	{attribute 'c++_compatible'}
	{attribute 'external_name' := 'FB_VN_ReadRegister_ULINT_GUID_0511260A_434E_4D8A_DC8D_C67C5FC0DC86'}
	{attribute 'TcIecLibraryType'}
	(* This FB reads a ULINT register from the camera. Requires an open control channel (e.g. by calling FB_VN_GevCameraControl.OpenCamera() before) *)
	FUNCTION_BLOCK FB_VN_ReadRegister_ULINT
	VAR_INPUT
		(* The address of the register that should be read *)
		 {attribute 'GUID' := 'E1ED2436-3512-43FA-B927-3F71DEDDA853'}
		nAddress : GVCP_REGISTER_ADDRESS;
		(* OPTIONAL: The endianness of the register. 0 = Big, 1 = Little. Default: 0 *)
		nEndian : UINT;
		(* Reading the register is triggered by a rising edge at this input. *)
		bRead : BOOL;
	END_VAR
	VAR
		 {attribute 'hide'}
		_reserved1 : USINT;
	END_VAR
	VAR_INPUT
		(* Indicates the time before the function is cancelled. *)
		nTimeout : TIME := VISION_ADS_TIMEOUT;
	END_VAR
	VAR
		 {attribute 'hide'}
		_reserved2 : UINT_0_32;
	END_VAR
	VAR_OUTPUT
		(* The read value *)
		nValue : ULINT;
		(* This output remains TRUE until the function block has executed a command, but at the longest for the duration supplied to the 'nTimeout' input. While bBusy = TRUE, no new command will be accepted at the inputs. *)
		bBusy : BOOL;
		(* This output is switched to TRUE as soon as an error occurs during the execution of a command. The command-specific error code is contained in ‘nErrorId’. If the function block has a timeout error, 'bError' is TRUE and 'nErrorId' is 1861 (hexadecimal 0x745). Is reset to FALSE by the execution of a command at the inputs. *)
		bError : BOOL;
	END_VAR
	VAR
		 {attribute 'hide'}
		_reserved3 : UINT;
	END_VAR
	VAR_OUTPUT
		(* Contains the ADS error code or the command-specific error code of the last executed command. Is reset to 0 by the execution of a command at the inputs. *)
		nErrorId : UDINT;
	END_VAR
	VAR
		(* Internal reference to the corresponding TcVnGevImageProvider TcCOM module ID, which needs to be set via TC init symbol. *)
		{attribute 'TcInitSymbol'}
		{attribute 'TcCategoryOID' := 'TcVnGevImageProvider'}
		 {attribute 'GUID' := '18071995-0000-0000-0000-00000000000F'}
		oidITcVnGevImageProvider : OTCID;
		 {attribute 'hide'}
		_reserved4 : UINT_0_32;
		(* Internal reference to the corresponding TcVnGevImageProvider module. *)
		{attribute 'hide'}
		 {attribute 'GUID' := 'ED7659DB-95DC-4A4A-B62F-02C9870D5E81'}
		ipGevImageProvider : ITcVnGevImageProvider;
		(* Internal timestamp for timeout detection *)
		{attribute 'hide'}
		nTimeElapsed : TIME;
		(* Internal flag for rising edge detection *)
		{attribute 'hide'}
		bLastRead : BOOL;
		 {attribute 'hide'}
		_reserved5 : ARRAY [1..3] OF USINT;
	END_VAR


	(* Internal method *)
	{attribute 'hide'}
	METHOD FB_exit : BOOL
	VAR_INPUT
		(*  if TRUE, the exit method is called for exiting an instance that is copied afterwards (online change). *)
		bInCopyCode : BOOL;
	END_VAR
END_METHOD


	(* Internal method *)
	{attribute 'hide'}
	METHOD FB_init : BOOL
	VAR_INPUT
		(*  if TRUE, the retain variables are initialized (warm start / cold start) *)
		bInitRetains : BOOL;
		(*  if TRUE, the instance afterwards gets moved into the copy code (online change) *)
		bInCopyCode : BOOL;
	END_VAR
END_METHOD

END_FUNCTION_BLOCK

// Function Blocks/Camera Register Access/FB_VN_WriteRegister_ULINT

	{attribute 'c++_compatible'}
	{attribute 'external_name' := 'FB_VN_WriteRegister_ULINT_GUID_9D472D1C_82B4_4199_F5A1_B64D0453F3B0'}
	{attribute 'TcIecLibraryType'}
	(* This FB writes a ULINT value into a register on the camera. Requires an open control channel (e.g. by calling FB_VN_GevCameraControl.OpenCamera() before) *)
	FUNCTION_BLOCK FB_VN_WriteRegister_ULINT
	VAR_INPUT
		(* The address of the register that should be written *)
		 {attribute 'GUID' := 'E1ED2436-3512-43FA-B927-3F71DEDDA853'}
		nAddress : GVCP_REGISTER_ADDRESS;
	END_VAR
	VAR
		 {attribute 'hide'}
		_reserved1 : UINT_0_32;
	END_VAR
	VAR_INPUT
		(* The value to write *)
		nValue : ULINT;
		(* OPTIONAL: The endianness of the register. 0 = Big, 1 = Little. Default: 0 *)
		nEndian : UINT;
		(* Writing the register is triggered by a rising edge at this input. *)
		bWrite : BOOL;
	END_VAR
	VAR
		 {attribute 'hide'}
		_reserved2 : USINT;
	END_VAR
	VAR_INPUT
		(* Indicates the time before the function is cancelled. *)
		nTimeout : TIME := VISION_ADS_TIMEOUT;
	END_VAR
	VAR_OUTPUT
		(* This output remains TRUE until the function block has executed a command, but at the longest for the duration supplied to the 'nTimeout' input. While bBusy = TRUE, no new command will be accepted at the inputs. *)
		bBusy : BOOL;
		(* This output is switched to TRUE as soon as an error occurs during the execution of a command. The command-specific error code is contained in ‘nErrorId’. If the function block has a timeout error, 'bError' is TRUE and 'nErrorId' is 1861 (hexadecimal 0x745). Is reset to FALSE by the execution of a command at the inputs. *)
		bError : BOOL;
	END_VAR
	VAR
		 {attribute 'hide'}
		_reserved3 : UINT;
	END_VAR
	VAR_OUTPUT
		(* Contains the ADS error code or the command-specific error code of the last executed command. Is reset to 0 by the execution of a command at the inputs. *)
		nErrorId : UDINT;
	END_VAR
	VAR
		(* Internal reference to the corresponding TcVnGevImageProvider TcCOM module ID, which needs to be set via TC init symbol. *)
		{attribute 'TcInitSymbol'}
		{attribute 'TcCategoryOID' := 'TcVnGevImageProvider'}
		 {attribute 'GUID' := '18071995-0000-0000-0000-00000000000F'}
		oidITcVnGevImageProvider : OTCID;
		 {attribute 'hide'}
		_reserved4 : UINT_0_32;
		(* Internal reference to the corresponding TcVnGevImageProvider module. *)
		{attribute 'hide'}
		 {attribute 'GUID' := 'ED7659DB-95DC-4A4A-B62F-02C9870D5E81'}
		ipGevImageProvider : ITcVnGevImageProvider;
		(* Internal timestamp for timeout detection *)
		{attribute 'hide'}
		nTimeElapsed : TIME;
		(* Internal flag for rising edge detection *)
		{attribute 'hide'}
		bLastWrite : BOOL;
		 {attribute 'hide'}
		_reserved5 : ARRAY [1..3] OF USINT;
	END_VAR


	(* Internal method *)
	{attribute 'hide'}
	METHOD FB_exit : BOOL
	VAR_INPUT
		(*  if TRUE, the exit method is called for exiting an instance that is copied afterwards (online change). *)
		bInCopyCode : BOOL;
	END_VAR
END_METHOD


	(* Internal method *)
	{attribute 'hide'}
	METHOD FB_init : BOOL
	VAR_INPUT
		(*  if TRUE, the retain variables are initialized (warm start / cold start) *)
		bInitRetains : BOOL;
		(*  if TRUE, the instance afterwards gets moved into the copy code (online change) *)
		bInCopyCode : BOOL;
	END_VAR
END_METHOD

END_FUNCTION_BLOCK

// Function Blocks/Camera Register Access/FB_VN_ReadMemory

	{attribute 'c++_compatible'}
	{attribute 'external_name' := 'FB_VN_ReadMemory_GUID_F43A0502_950A_4FC1_EE1B_7AC9DA03F230'}
	{attribute 'TcIecLibraryType'}
	(* This FB reads consecutive memory locations from the camera. Requires an open control channel (e.g. by calling FB_VN_GevCameraControl.OpenCamera() before) *)
	FUNCTION_BLOCK FB_VN_ReadMemory
	VAR_INPUT
		(* The address of the first byte to read from the camera (must be 32-bit aligned) *)
		 {attribute 'GUID' := 'E1ED2436-3512-43FA-B927-3F71DEDDA853'}
		nAddress : GVCP_REGISTER_ADDRESS;
		(* The number of bytes to read, starting with nAddress (must be a multiple of 4, not more than 536) *)
		nLength : UINT;
	END_VAR
	VAR
		 {attribute 'hide'}
		_reserved1 : UINT;
	END_VAR
	VAR_INPUT
		(* Pointer to the buffer where the read memory content is written to (The buffer must have a size of at least nLength bytes!) *)
		 {attribute 'GUID' := '18071995-0000-0000-0000-000000000018'}
		pBuffer : PVOID;
		(* Reading the memory is triggered by a rising edge at this input. *)
		bRead : BOOL;
	END_VAR
	VAR
		 {attribute 'hide'}
		_reserved2 : ARRAY [1..3] OF USINT;
	END_VAR
	VAR_INPUT
		(* Indicates the time before the function is cancelled. *)
		nTimeout : TIME := VISION_ADS_TIMEOUT;
	END_VAR
	VAR_OUTPUT
		(* This output remains TRUE until the function block has executed a command, but at the longest for the duration supplied to the 'nTimeout' input. While bBusy = TRUE, no new command will be accepted at the inputs. *)
		bBusy : BOOL;
		(* This output is switched to TRUE as soon as an error occurs during the execution of a command. The command-specific error code is contained in ‘nErrorId’. If the function block has a timeout error, 'bError' is TRUE and 'nErrorId' is 1861 (hexadecimal 0x745). Is reset to FALSE by the execution of a command at the inputs. *)
		bError : BOOL;
	END_VAR
	VAR
		 {attribute 'hide'}
		_reserved3 : UINT;
	END_VAR
	VAR_OUTPUT
		(* Contains the ADS error code or the command-specific error code of the last executed command. Is reset to 0 by the execution of a command at the inputs. *)
		nErrorId : UDINT;
	END_VAR
	VAR
		(* Internal reference to the corresponding TcVnGevImageProvider TcCOM module ID, which needs to be set via TC init symbol. *)
		{attribute 'TcInitSymbol'}
		{attribute 'TcCategoryOID' := 'TcVnGevImageProvider'}
		 {attribute 'GUID' := '18071995-0000-0000-0000-00000000000F'}
		oidITcVnGevImageProvider : OTCID;
		 {attribute 'hide'}
		_reserved4 : UINT_0_32;
		(* Internal reference to the corresponding TcVnGevImageProvider module. *)
		{attribute 'hide'}
		 {attribute 'GUID' := 'ED7659DB-95DC-4A4A-B62F-02C9870D5E81'}
		ipGevImageProvider : ITcVnGevImageProvider;
		(* Internal timestamp for timeout detection *)
		{attribute 'hide'}
		nTimeElapsed : TIME;
		(* Internal flag for rising edge detection *)
		{attribute 'hide'}
		bLastRead : BOOL;
		 {attribute 'hide'}
		_reserved5 : ARRAY [1..3] OF USINT;
	END_VAR


	(* Internal method *)
	{attribute 'hide'}
	METHOD FB_exit : BOOL
	VAR_INPUT
		(* If TRUE, the exit method is called for exiting an instance that is copied afterwards (online change). *)
		bInCopyCode : BOOL;
	END_VAR
END_METHOD


	(* Internal method *)
	{attribute 'hide'}
	METHOD FB_init : BOOL
	VAR_INPUT
		(* If TRUE, the retain variables are initialized (warm start / cold start) *)
		bInitRetains : BOOL;
		(* If TRUE, the instance afterwards gets moved into the copy code (online change) *)
		bInCopyCode : BOOL;
	END_VAR
END_METHOD

END_FUNCTION_BLOCK

// Function Blocks/Camera Register Access/FB_VN_WriteMemory

	{attribute 'c++_compatible'}
	{attribute 'external_name' := 'FB_VN_WriteMemory_GUID_E11A1718_DC13_44E5_FD90_B3F294477065'}
	{attribute 'TcIecLibraryType'}
	(* This FB writes data to consecutive memory locations on the camera. Requires an open control channel (e.g. by calling FB_VN_GevCameraControl.OpenCamera() before) *)
	FUNCTION_BLOCK FB_VN_WriteMemory
	VAR_INPUT
		(* The address of the first byte to write to the camera (must be 32-bit aligned) *)
		 {attribute 'GUID' := 'E1ED2436-3512-43FA-B927-3F71DEDDA853'}
		nAddress : GVCP_REGISTER_ADDRESS;
		(* The number of bytes to write, starting at nAddress (must be a multiple of 4, not more than 536) *)
		nLength : UINT;
	END_VAR
	VAR
		 {attribute 'hide'}
		_reserved1 : UINT;
	END_VAR
	VAR_INPUT
		(* Pointer to the data that should be written to the camera (must have a size of at least nLength bytes!) *)
		 {attribute 'GUID' := '18071995-0000-0000-0000-000000000018'}
		pData : PVOID;
		(* Writing the memory is triggered by a rising edge at this input. *)
		bWrite : BOOL;
	END_VAR
	VAR
		 {attribute 'hide'}
		_reserved2 : ARRAY [1..3] OF USINT;
	END_VAR
	VAR_INPUT
		(* Indicates the time before the function is cancelled. *)
		nTimeout : TIME := VISION_ADS_TIMEOUT;
	END_VAR
	VAR_OUTPUT
		(* This output remains TRUE until the function block has executed a command, but at the longest for the duration supplied to the 'nTimeout' input. While bBusy = TRUE, no new command will be accepted at the inputs. *)
		bBusy : BOOL;
		(* This output is switched to TRUE as soon as an error occurs during the execution of a command. The command-specific error code is contained in ‘nErrorId’. If the function block has a timeout error, 'bError' is TRUE and 'nErrorId' is 1861 (hexadecimal 0x745). Is reset to FALSE by the execution of a command at the inputs. *)
		bError : BOOL;
	END_VAR
	VAR
		 {attribute 'hide'}
		_reserved3 : UINT;
	END_VAR
	VAR_OUTPUT
		(* Contains the ADS error code or the command-specific error code of the last executed command. Is reset to 0 by the execution of a command at the inputs. *)
		nErrorId : UDINT;
		(* The number of bytes that have been successfully written to the camera. *)
		nBytesWritten : UINT;
	END_VAR
	VAR
		 {attribute 'hide'}
		_reserved4 : UINT;
		(* Internal reference to the corresponding TcVnGevImageProvider TcCOM module ID, which needs to be set via TC init symbol. *)
		{attribute 'TcInitSymbol'}
		{attribute 'TcCategoryOID' := 'TcVnGevImageProvider'}
		 {attribute 'GUID' := '18071995-0000-0000-0000-00000000000F'}
		oidITcVnGevImageProvider : OTCID;
		(* Internal reference to the corresponding TcVnGevImageProvider module. *)
		{attribute 'hide'}
		 {attribute 'GUID' := 'ED7659DB-95DC-4A4A-B62F-02C9870D5E81'}
		ipGevImageProvider : ITcVnGevImageProvider;
		(* Internal timestamp for timeout detection *)
		{attribute 'hide'}
		nTimeElapsed : TIME;
		(* Internal flag for rising edge detection *)
		{attribute 'hide'}
		bLastRead : BOOL;
		 {attribute 'hide'}
		_reserved5 : ARRAY [1..3] OF USINT;
	END_VAR


	(* Internal method *)
	{attribute 'hide'}
	METHOD FB_exit : BOOL
	VAR_INPUT
		(* If TRUE, the exit method is called for exiting an instance that is copied afterwards (online change). *)
		bInCopyCode : BOOL;
	END_VAR
END_METHOD


	(* Internal method *)
	{attribute 'hide'}
	METHOD FB_init : BOOL
	VAR_INPUT
		(* If TRUE, the retain variables are initialized (warm start / cold start) *)
		bInitRetains : BOOL;
		(* If TRUE, the instance afterwards gets moved into the copy code (online change) *)
		bInCopyCode : BOOL;
	END_VAR
END_METHOD

END_FUNCTION_BLOCK

// Function Blocks/Camera Register Access/FB_VN_ReadRegister_REAL

	{attribute 'c++_compatible'}
	{attribute 'external_name' := 'FB_VN_ReadRegister_REAL_GUID_8300240C_129D_40AD_E145_72F0B3958AC0'}
	{attribute 'TcIecLibraryType'}
	(* This FB reads a REAL register from the camera. Requires an open control channel (e.g. by calling FB_VN_GevCameraControl.OpenCamera() before) *)
	FUNCTION_BLOCK FB_VN_ReadRegister_REAL
	VAR_INPUT
		(* The address of the register that should be read *)
		 {attribute 'GUID' := 'E1ED2436-3512-43FA-B927-3F71DEDDA853'}
		nAddress : GVCP_REGISTER_ADDRESS;
		(* OPTIONAL: The endianness of the register. 0 = Big, 1 = Little. Default: 0 *)
		nEndian : UINT;
		(* Reading the register is triggered by a rising edge at this input. *)
		bRead : BOOL;
	END_VAR
	VAR
		 {attribute 'hide'}
		_reserved1 : USINT;
	END_VAR
	VAR_INPUT
		(* Indicates the time before the function is cancelled. *)
		nTimeout : TIME := VISION_ADS_TIMEOUT;
	END_VAR
	VAR_OUTPUT
		(* The read value *)
		fValue : REAL;
		(* This output remains TRUE until the function block has executed a command, but at the longest for the duration supplied to the 'nTimeout' input. While bBusy = TRUE, no new command will be accepted at the inputs. *)
		bBusy : BOOL;
		(* This output is switched to TRUE as soon as an error occurs during the execution of a command. The command-specific error code is contained in ‘nErrorId’. If the function block has a timeout error, 'bError' is TRUE and 'nErrorId' is 1861 (hexadecimal 0x745). Is reset to FALSE by the execution of a command at the inputs. *)
		bError : BOOL;
	END_VAR
	VAR
		 {attribute 'hide'}
		_reserved2 : UINT;
	END_VAR
	VAR_OUTPUT
		(* Contains the ADS error code or the command-specific error code of the last executed command. Is reset to 0 by the execution of a command at the inputs. *)
		nErrorId : UDINT;
	END_VAR
	VAR
		(* Internal reference to the corresponding TcVnGevImageProvider TcCOM module ID, which needs to be set via TC init symbol. *)
		{attribute 'TcInitSymbol'}
		{attribute 'TcCategoryOID' := 'TcVnGevImageProvider'}
		 {attribute 'GUID' := '18071995-0000-0000-0000-00000000000F'}
		oidITcVnGevImageProvider : OTCID;
		 {attribute 'hide'}
		_reserved3 : UINT_0_32;
		(* Internal reference to the corresponding TcVnGevImageProvider module. *)
		{attribute 'hide'}
		 {attribute 'GUID' := 'ED7659DB-95DC-4A4A-B62F-02C9870D5E81'}
		ipGevImageProvider : ITcVnGevImageProvider;
		(* Internal timestamp for timeout detection *)
		{attribute 'hide'}
		nTimeElapsed : TIME;
		(* Internal flag for rising edge detection *)
		{attribute 'hide'}
		bLastRead : BOOL;
		 {attribute 'hide'}
		_reserved4 : ARRAY [1..3] OF USINT;
	END_VAR


	(* Internal method *)
	{attribute 'hide'}
	METHOD FB_exit : BOOL
	VAR_INPUT
		(*  if TRUE, the exit method is called for exiting an instance that is copied afterwards (online change). *)
		bInCopyCode : BOOL;
	END_VAR
END_METHOD


	(* Internal method *)
	{attribute 'hide'}
	METHOD FB_init : BOOL
	VAR_INPUT
		(*  if TRUE, the retain variables are initialized (warm start / cold start) *)
		bInitRetains : BOOL;
		(*  if TRUE, the instance afterwards gets moved into the copy code (online change) *)
		bInCopyCode : BOOL;
	END_VAR
END_METHOD

END_FUNCTION_BLOCK

// Function Blocks/Camera Register Access/FB_VN_WriteRegister_REAL

	{attribute 'c++_compatible'}
	{attribute 'external_name' := 'FB_VN_WriteRegister_REAL_GUID_9406F075_95E1_49DE_E4AE_6ECDFB627AD5'}
	{attribute 'TcIecLibraryType'}
	(* This FB writes a REAL value into a register on the camera. Requires an open control channel (e.g. by calling FB_VN_GevCameraControl.OpenCamera() before) *)
	FUNCTION_BLOCK FB_VN_WriteRegister_REAL
	VAR_INPUT
		(* The address of the register that should be written *)
		 {attribute 'GUID' := 'E1ED2436-3512-43FA-B927-3F71DEDDA853'}
		nAddress : GVCP_REGISTER_ADDRESS;
		(* The value to write *)
		fValue : REAL;
		(* OPTIONAL: The endianness of the register. 0 = Big, 1 = Little. Default: 0 *)
		nEndian : UINT;
		(* Writing the register is triggered by a rising edge at this input. *)
		bWrite : BOOL;
	END_VAR
	VAR
		 {attribute 'hide'}
		_reserved1 : USINT;
	END_VAR
	VAR_INPUT
		(* Indicates the time before the function is cancelled. *)
		nTimeout : TIME := VISION_ADS_TIMEOUT;
	END_VAR
	VAR_OUTPUT
		(* This output remains TRUE until the function block has executed a command, but at the longest for the duration supplied to the 'nTimeout' input. While bBusy = TRUE, no new command will be accepted at the inputs. *)
		bBusy : BOOL;
		(* This output is switched to TRUE as soon as an error occurs during the execution of a command. The command-specific error code is contained in ‘nErrorId’. If the function block has a timeout error, 'bError' is TRUE and 'nErrorId' is 1861 (hexadecimal 0x745). Is reset to FALSE by the execution of a command at the inputs. *)
		bError : BOOL;
	END_VAR
	VAR
		 {attribute 'hide'}
		_reserved2 : UINT;
	END_VAR
	VAR_OUTPUT
		(* Contains the ADS error code or the command-specific error code of the last executed command. Is reset to 0 by the execution of a command at the inputs. *)
		nErrorId : UDINT;
	END_VAR
	VAR
		(* Internal reference to the corresponding TcVnGevImageProvider TcCOM module ID, which needs to be set via TC init symbol. *)
		{attribute 'TcInitSymbol'}
		{attribute 'TcCategoryOID' := 'TcVnGevImageProvider'}
		 {attribute 'GUID' := '18071995-0000-0000-0000-00000000000F'}
		oidITcVnGevImageProvider : OTCID;
		 {attribute 'hide'}
		_reserved3 : UINT_0_32;
		(* Internal reference to the corresponding TcVnGevImageProvider module. *)
		{attribute 'hide'}
		 {attribute 'GUID' := 'ED7659DB-95DC-4A4A-B62F-02C9870D5E81'}
		ipGevImageProvider : ITcVnGevImageProvider;
		(* Internal timestamp for timeout detection *)
		{attribute 'hide'}
		nTimeElapsed : TIME;
		(* Internal flag for rising edge detection *)
		{attribute 'hide'}
		bLastWrite : BOOL;
		 {attribute 'hide'}
		_reserved4 : ARRAY [1..3] OF USINT;
	END_VAR


	(* Internal method *)
	{attribute 'hide'}
	METHOD FB_exit : BOOL
	VAR_INPUT
		(*  if TRUE, the exit method is called for exiting an instance that is copied afterwards (online change). *)
		bInCopyCode : BOOL;
	END_VAR
END_METHOD


	(* Internal method *)
	{attribute 'hide'}
	METHOD FB_init : BOOL
	VAR_INPUT
		(*  if TRUE, the retain variables are initialized (warm start / cold start) *)
		bInitRetains : BOOL;
		(*  if TRUE, the instance afterwards gets moved into the copy code (online change) *)
		bInCopyCode : BOOL;
	END_VAR
END_METHOD

END_FUNCTION_BLOCK

// Function Blocks/Image Processing/FB_VN_GeneralizedHoughBallard

	{attribute 'c++_compatible'}
	{attribute 'external_name' := 'FB_VN_GeneralizedHoughBallard_GUID_A0476776_FAE7_4198_C858_300BFA209DB8'}
	{attribute 'TcIecLibraryType'}
	{attribute 'no_explicit_call' :='do not call this POU directly'}
	(* This FB provides the Generalized Hough Ballard functionality. First, set the parameters via the corresponding methods (optional, defaults are used otherwise). Then, set the template (required). Afterwards, the Detect method can be executed. *)
	FUNCTION_BLOCK FB_VN_GeneralizedHoughBallard
	VAR
		(* Internal stuff *)
		{attribute 'hide'}
		 {attribute 'GUID' := '18071995-0000-0000-0000-000000000018'}
		internal1 : PVOID;
		(* Internal stuff *)
		{attribute 'hide'}
		 {attribute 'GUID' := '18071995-0000-0000-0000-000000000018'}
		internal2 : PVOID;
		(* Internal stuff *)
		{attribute 'hide'}
		internal3 : BOOL;
		 {attribute 'hide'}
		_reserved1 : UINT_24_56;
	END_VAR


	(* Internal method *)
	{attribute 'hide'}
	METHOD FB_exit : BOOL
	VAR_INPUT
		(* if TRUE, the exit method is called for exiting an instance that is copied afterwards (online change). *)
		bInCopyCode : BOOL;
	END_VAR
END_METHOD


	(* Internal method *)
	{attribute 'hide'}
	METHOD FB_init : BOOL
	VAR_INPUT
		(* if TRUE, the retain variables are initialized (warm start / cold start) *)
		bInitRetains : BOOL;
		(* if TRUE, the instance afterwards gets moved into the copy code (online change) *)
		bInCopyCode : BOOL;
	END_VAR
END_METHOD


	(* Detect the template in an image (SetTemplate must have been called before). *)
	METHOD Detect : HRESULT
	VAR_INPUT
		(* Source image (1 channel, USINT) *)
 {attribute 'GUID' := '70D42C6D-6F4E-4719-8B29-2883D5D59B1C'}
				ipImage : ITcVnImage;
		(* Returns the centers of the detected template positions (ContainerType_Vector_TcVnPoint2_REAL; Non-zero interface pointers are reused.) *)
 {attribute 'GUID' := 'BC72B333-E095-465B-9693-7979773CA3B8'}
				ipPositions : REFERENCE TO ITcVnContainer;
	END_VAR
END_METHOD


	(* Sets the canny edge detection thresholds. *)
	METHOD SetCannyThreshold : HRESULT
	VAR_INPUT
		(* Low threshold (> 0) *)
		nLow : DINT;
		(* High threshold (> nLow, usually 2 to 3 * nLow) *)
		nHigh : DINT;
	END_VAR
END_METHOD


	(* Sets the inverted ratio of the accumulator size in relation to the source image's size (e.g. a value of 2 means that the size is halved in both directions.) *)
	METHOD SetInvAccuRatio : HRESULT
	VAR_INPUT
		(* Inverted accumulator ratio (> 0) *)
		fInvAccuRatio : LREAL;
	END_VAR
END_METHOD


	(* Sets the number of R-table levels. *)
	METHOD SetLevels : HRESULT
	VAR_INPUT
		(* Number of R-table levels (> 0) *)
		nLevels : DINT;
	END_VAR
END_METHOD


	(* Sets the minimum distance between the centers of different objects. *)
	METHOD SetMinDist : HRESULT
	VAR_INPUT
		(* Minimum distance (> 0) *)
		fMinDist : LREAL;
	END_VAR
END_METHOD


	(* Sets the template image to search for in the Detect method. *)
	METHOD SetTemplate : HRESULT
	VAR_INPUT
		(* Template image (1 channel, USINT) *)
 {attribute 'GUID' := '70D42C6D-6F4E-4719-8B29-2883D5D59B1C'}
				ipImage : ITcVnImage;
	END_VAR
END_METHOD


	(* Sets the accumulator threshold, i.e. the number of votes required to detect a match (too small values lead to false detections). *)
	METHOD SetVotesThreshold : HRESULT
	VAR_INPUT
		(* Number of votes required to detect a match (> 0) *)
		nVotes : DINT;
	END_VAR
END_METHOD

END_FUNCTION_BLOCK

// Function Blocks/Image Processing/FB_VN_SSIM

	{attribute 'c++_compatible'}
	{attribute 'external_name' := 'FB_VN_SSIM_GUID_4075B8D8_49BB_4B5C_CD74_E48AAA73AD77'}
	{attribute 'TcIecLibraryType'}
	{attribute 'no_explicit_call' :='do not call this POU directly'}
	(* This FB provides the structural similarity (SSIM) functionality. First, set the reference image. Afterwards, the Compute method can be executed. *)
	FUNCTION_BLOCK FB_VN_SSIM
	VAR
		(* Internal stuff *)
		{attribute 'hide'}
		 {attribute 'GUID' := '18071995-0000-0000-0000-000000000018'}
		internal1 : PVOID;
	END_VAR


	(* Internal method *)
	{attribute 'hide'}
	METHOD FB_exit : BOOL
	VAR_INPUT
		(* if TRUE, the exit method is called for exiting an instance that is copied afterwards (online change). *)
		bInCopyCode : BOOL;
	END_VAR
END_METHOD


	(* Internal method *)
	{attribute 'hide'}
	METHOD FB_init : BOOL
	VAR_INPUT
		(* if TRUE, the retain variables are initialized (warm start / cold start) *)
		bInitRetains : BOOL;
		(* if TRUE, the instance afterwards gets moved into the copy code (online change) *)
		bInCopyCode : BOOL;
	END_VAR
END_METHOD


	(* Compute the structural similarity (SetReference must have been called before). *)
	METHOD Compute : HRESULT
	VAR_INPUT
		(* Source image (USINT) *)
 {attribute 'GUID' := '70D42C6D-6F4E-4719-8B29-2883D5D59B1C'}
				ipSrcImage : ITcVnImage;
		(* Returns the SSIM (REAL, values from 0 to 1) *)
 {attribute 'GUID' := '70D42C6D-6F4E-4719-8B29-2883D5D59B1C'}
				ipSSIM : REFERENCE TO ITcVnImage;
	END_VAR
END_METHOD


	(* Sets the reference image, used by the SSIM method. *)
	METHOD SetReference : HRESULT
	VAR_INPUT
		(* Reference image (USINT) *)
 {attribute 'GUID' := '70D42C6D-6F4E-4719-8B29-2883D5D59B1C'}
				ipImage : ITcVnImage;
	END_VAR
END_METHOD

END_FUNCTION_BLOCK

// Functions/Control Functions/F_VN_StartAbsWatchdog

	{attribute 'TcIecLibraryType'}
	{attribute 'external_name' := 'F_VN_StartAbsWatchdog_GUID_354F303E_246D_4234_D496_3202655F920B'}
	(* Starts a cooperative watchdog given an absolute stop time. *)
	FUNCTION F_VN_StartAbsWatchdog : HRESULT
	VAR_INPUT
		tStop	:	DINT;	(* Stop time in us *)
		hrPrev	:	HRESULT;	(* HRESULT indicating the result of previous operations (If SUCCEEDED(hrPrev) equals false, no operation is executed.) *)
	END_VAR

END_FUNCTION

// Functions/Control Functions/F_VN_StartAbsWatchdogExp

	{attribute 'TcIecLibraryType'}
	{attribute 'external_name' := 'F_VN_StartAbsWatchdogExp_GUID_A505C06B_6324_4EA0_F923_AC5477E9F7DD'}
	(* Start a cooperative watchdog given an absolute stop time. (expert function) *)
	FUNCTION F_VN_StartAbsWatchdogExp : HRESULT
	VAR_INPUT
		tStop	:	DINT;	(* Stop time in us *)
		eWatchdogAccType	:	ETcWatchdogAccumulationType;	(* Accumalation method used for combining the results of multiple functions enclosed by this watchdog *)
		hrPrev	:	HRESULT;	(* HRESULT indicating the result of previous operations (If SUCCEEDED(hrPrev) equals false, no operation is executed.) *)
	END_VAR

END_FUNCTION

// Functions/Control Functions/F_VN_StartRelWatchdog

	{attribute 'TcIecLibraryType'}
	{attribute 'external_name' := 'F_VN_StartRelWatchdog_GUID_CECC2BA7_165D_4C64_F30F_7230AFEEB944'}
	(* Starts a cooperative watchdog given a stop time relative to the current time. *)
	FUNCTION F_VN_StartRelWatchdog : HRESULT
	VAR_INPUT
		tStop	:	DINT;	(* Stop time in us *)
		hrPrev	:	HRESULT;	(* HRESULT indicating the result of previous operations (If SUCCEEDED(hrPrev) equals false, no operation is executed.) *)
	END_VAR

END_FUNCTION

// Functions/Control Functions/F_VN_StartRelWatchdogExp

	{attribute 'TcIecLibraryType'}
	{attribute 'external_name' := 'F_VN_StartRelWatchdogExp_GUID_CD8CE6D1_94FB_4654_D6A0_F6BBAA9F615D'}
	(* Start a cooperative watchdog given a stop time relative to the current time. (expert function) *)
	FUNCTION F_VN_StartRelWatchdogExp : HRESULT
	VAR_INPUT
		tStop	:	DINT;	(* Stop time in us *)
		eWatchdogAccType	:	ETcWatchdogAccumulationType;	(* Accumalation method used for combining the results of multiple functions enclosed by this watchdog *)
		hrPrev	:	HRESULT;	(* HRESULT indicating the result of previous operations (If SUCCEEDED(hrPrev) equals false, no operation is executed.) *)
	END_VAR

END_FUNCTION

// Functions/Control Functions/F_VN_StopWatchdog

	{attribute 'TcIecLibraryType'}
	{attribute 'external_name' := 'F_VN_StopWatchdog_GUID_A7144577_78C6_4DD5_EF4C_E05E8BBCA2CE'}
	(* Stops a watchdog and provide runtime information. *)
	FUNCTION F_VN_StopWatchdog : HRESULT
	VAR_INPUT
		hrStartWatchdog	:	HRESULT;	(* HRESULT indicating the result of the function used to start the watchdog (If SUCCEEDED(hrStartWatchdog) equals false, no operation is executed.) *)
	END_VAR
	VAR_OUTPUT
		nFunctionsMonitored	:	ULINT;	(* Returns the number of functions monitored *)
		nFractionProcessed	:	UDINT;	(* Returns the fraction processed accumulated over the monitored functions in percent *)
		tRest	:	DINT;	(* Returns the remaining computation time in us (may be negative) *)
	END_VAR

END_FUNCTION

// Functions/Image Segmentation/F_VN_AdaptiveThreshold

	{attribute 'TcIecLibraryType'}
	{attribute 'external_name' := 'F_VN_AdaptiveThreshold_GUID_49401DDC_F3BE_44F8_E05C_C9E83DEAC857'}
	(* Apply an adaptive threshold to a gray level image. *)
	FUNCTION F_VN_AdaptiveThreshold : HRESULT
	VAR_INPUT
		ipSrcImage	:	ITcVnImage;	(* Source image (1 channel, elements of type USINT) *)
		ipDestImage	:	REFERENCE TO ITcVnImage;	(* Destination image (An appropriate destination image will be created if required.) *)
		fMaxValue	:	LREAL;	(* Value assigned to pixels for which the threshold condition is true *)
		hrPrev	:	HRESULT;	(* HRESULT indicating the result of previous operations (If SUCCEEDED(hrPrev) equals false, no operation is executed.) *)
	END_VAR

END_FUNCTION

// Functions/Image Segmentation/F_VN_AdaptiveThresholdExp

	{attribute 'TcIecLibraryType'}
	{attribute 'external_name' := 'F_VN_AdaptiveThresholdExp_GUID_1CE298F0_0C53_40FE_E76E_6A320A21FB73'}
	(* Apply an adaptive threshold to a gray level image. (expert function) *)
	FUNCTION F_VN_AdaptiveThresholdExp : HRESULT
	VAR_INPUT
		ipSrcImage	:	ITcVnImage;	(* Source image (1 channel, elements of type USINT) *)
		ipDestImage	:	REFERENCE TO ITcVnImage;	(* Destination image (An appropriate destination image will be created if required.) *)
		fMaxValue	:	LREAL;	(* Value assigned to pixels for which the threshold condition is true *)
		eAdaptiveMethod	:	ETcVnAdaptiveThresholdMethod;	(* Adaptive threshold method to be applied (MEAN: threshold value will be calculated as a mean of the nBlockSize x nBlockSize neighborhood of (x,y) minus fConstant. GAUSSIAN: threshold value is a weighted sum (cross-correlation with a Gaussian window) of the nBlockSize x nBlockSize neighborhood of (x,y) minus fConstant. *)
		eThresholdType	:	ETcVnThresholdType;	(* Threshold type to be applied (only BINARY and BINARY_INV are supported) *)
		nBlockSize	:	UDINT;	(* Size of the pixel neighborhood to calculate the local threshold (3, 5, 7, ...) *)
		fConstant	:	LREAL;	(* Constant that is subtracted from the weighted mean of the pixel neighborhood, which leads to the local threshold *)
		hrPrev	:	HRESULT;	(* HRESULT indicating the result of previous operations (If SUCCEEDED(hrPrev) equals false, no operation is executed.) *)
	END_VAR

END_FUNCTION

// Functions/Image Segmentation/F_VN_CheckColorRange

	{attribute 'TcIecLibraryType'}
	{attribute 'external_name' := 'F_VN_CheckColorRange_GUID_A7F9F0B9_4809_4E55_F379_CF12FF23991F'}
	(* Check if the pixel values of an image lie in a given range. The destination image has the same size as the source image but only one channel with
          a pixel element size of 8 bit. Its elements are set to 255 if the corresponding pixels of the source image are in the checked range and set to 0 otherwise. *)
	FUNCTION F_VN_CheckColorRange : HRESULT
	VAR_INPUT
		ipSrcImage	:	ITcVnImage;	(* Source image *)
		ipDestImage	:	REFERENCE TO ITcVnImage;	(* Destination image (An appropriate destination image will be created if required.) *)
	END_VAR
	VAR_IN_OUT
		aLowerBounds	:	TcVnVector4_LREAL;	(* Channel-wise lower bounds (Unused channels are ignored.) *)
		aUpperBounds	:	TcVnVector4_LREAL;	(* Channel-wise upper bounds (Unused channels are ignored.) *)
	END_VAR
	VAR_INPUT
		hrPrev	:	HRESULT;	(* HRESULT indicating the result of previous operations (If SUCCEEDED(hrPrev) equals false, no operation is executed.) *)
	END_VAR

END_FUNCTION

// Functions/Image Segmentation/F_VN_DoubleThreshold

	{attribute 'TcIecLibraryType'}
	{attribute 'external_name' := 'F_VN_DoubleThreshold_GUID_80CBDA5D_FA99_485A_F7EC_4F18E01B8AFC'}
	(* Apply a double threshold (also called hysteresis threshold) using morphological reconstruction. *)
	FUNCTION F_VN_DoubleThreshold : HRESULT
	VAR_INPUT
		ipSrcImage	:	ITcVnImage;	(* Source image (USINT, UINT, INT, REAL, or LREAL, 1 channel) *)
		ipDestImage	:	REFERENCE TO ITcVnImage;	(* Destination image (An appropriate destination image will be created if required.) *)
		fLowThreshold	:	LREAL;	(* Low threshold determinining the shape of found regions *)
		fHighThreshold	:	LREAL;	(* High threshold selecting found regions (Each region must at least contain a single pixel if the high threshold is applied.) *)
		fMaxValue	:	LREAL;	(* Maximum pixel value *)
		hrPrev	:	HRESULT;	(* HRESULT indicating the result of previous operations (If SUCCEEDED(hrPrev) equals false, no operation is executed.) *)
	END_VAR

END_FUNCTION

// Functions/Image Segmentation/F_VN_SauvolaThreshold

	{attribute 'TcIecLibraryType'}
	{attribute 'external_name' := 'F_VN_SauvolaThreshold_GUID_876189B7_ACAD_4F38_E000_3EC7AB409032'}
	(* Apply Sauvola local threshold to source image. *)
	FUNCTION F_VN_SauvolaThreshold : HRESULT
	VAR_INPUT
		ipSrcImage	:	ITcVnImage;	(* Source image (USINT, UINT, INT, REAL, or LREAL, 1 channel) *)
		pipDestImage	:	REFERENCE TO ITcVnImage;	(* Destination image (An appropriate single channel destination image will be created if required.)) *)
		nBlockSize	:	UDINT;	(* Size of the pixel neighborhood to calculate the local threshold (3, 5, 7, ...) *)
		fParamK	:	LREAL;	(* parameter K which takes positive values in range (0,1). Recommended are K in range [0.2, 0.5] *)
		fMaxSigma	:	LREAL;	(* Maximum value of the standard deviation, required to be strictly positive. (fMaxSigma = 128 for a grayscale document).   *)
		eThresholdType	:	ETcVnThresholdType;	(* Threshold type to be applied. Supported are TCVN_TT_BINARY and TCVN_TT_BINARY_INV. *)
		hrPrev	:	HRESULT;	(* HRESULT indicating the result of previous operations (If SUCCEEDED(hrPrev) equals false, no operation is executed.) *)
	END_VAR

END_FUNCTION

// Functions/Image Segmentation/F_VN_Threshold

	{attribute 'TcIecLibraryType'}
	{attribute 'external_name' := 'F_VN_Threshold_GUID_0C43ECB3_121B_4F58_D75E_64B84E1B47B2'}
	(* Apply a fixed threshold or a dynamic threshold according to Otsu. *)
	FUNCTION F_VN_Threshold : HRESULT
	VAR_INPUT
		ipSrcImage	:	ITcVnImage;	(* Source image (For Otsu and Triangle threshold types, only 1 channel of TCVN_ET_USINT is supported) *)
		ipDestImage	:	REFERENCE TO ITcVnImage;	(* Destination image (An appropriate destination image will be created if required.) *)
		fThreshold	:	LREAL;	(* Fixed threshold (unused if dynamic thresholding is selected) *)
		fMaxValue	:	LREAL;	(* Maximum pixel value *)
		eThresholdType	:	ETcVnThresholdType;	(* Threshold type to be applied *)
		hrPrev	:	HRESULT;	(* HRESULT indicating the result of previous operations (If SUCCEEDED(hrPrev) equals false, no operation is executed.) *)
	END_VAR

END_FUNCTION

// Functions/Image Segmentation/F_VN_WatershedSegmentationExp

	{attribute 'TcIecLibraryType'}
	{attribute 'external_name' := 'F_VN_WatershedSegmentationExp_GUID_FDB829B0_9CA2_4473_D9E8_89903FC44F81'}
	(* Apply a marker-based watershed segmentation. (expert function) *)
	FUNCTION F_VN_WatershedSegmentationExp : HRESULT
	VAR_INPUT
		ipSrcImage	:	ITcVnImage;	(* Source image (USINT, 3 channels) *)
		ipDestImage	:	REFERENCE TO ITcVnImage;	(* Destination image (DINT, 1 channel. An appropriate image will be created if required.) *)
		ipMarkers	:	ITcVnImage;	(* Marker image (DINT, 1 channel) *)
		hrPrev	:	HRESULT;	(* HRESULT indicating the result of previous operations (If SUCCEEDED(hrPrev) equals false, no operation is executed.) *)
	END_VAR

END_FUNCTION

// Functions/Algebraic Container Operations/F_VN_AddContainers

	{attribute 'TcIecLibraryType'}
	{attribute 'external_name' := 'F_VN_AddContainers_GUID_CC340976_D13B_4FF4_E209_5F431B9D653B'}
	(* Element-wise addition of two containers (same length and type). *)
	FUNCTION F_VN_AddContainers : HRESULT
	VAR_INPUT
		ipSrcContainer1	:	ITcVnContainer;	(* Source container 1 *)
		ipSrcContainer2	:	ITcVnContainer;	(* Source container 2 *)
		ipDestContainer	:	REFERENCE TO ITcVnContainer;	(* Returns the resulting container *)
		hrPrev	:	HRESULT;	(* HRESULT indicating the result of previous operations (If SUCCEEDED(hrPrev) equals false, no operation is executed.) *)
	END_VAR

END_FUNCTION

// Functions/Algebraic Container Operations/F_VN_BitwiseAndContainers

	{attribute 'TcIecLibraryType'}
	{attribute 'external_name' := 'F_VN_BitwiseAndContainers_GUID_138910BC_F79B_4F2A_F3AC_89E247834407'}
	(* Element-wise application of a bit-wise AND operator to two containers (same length and type, integer only). *)
	FUNCTION F_VN_BitwiseAndContainers : HRESULT
	VAR_INPUT
		ipSrcContainer1	:	ITcVnContainer;	(* Source container 1 *)
		ipSrcContainer2	:	ITcVnContainer;	(* Source container 2 *)
		ipDestContainer	:	REFERENCE TO ITcVnContainer;	(* Returns the resulting container *)
		hrPrev	:	HRESULT;	(* HRESULT indicating the result of previous operations (If SUCCEEDED(hrPrev) equals false, no operation is executed.) *)
	END_VAR

END_FUNCTION

// Functions/Algebraic Container Operations/F_VN_BitwiseNotContainer

	{attribute 'TcIecLibraryType'}
	{attribute 'external_name' := 'F_VN_BitwiseNotContainer_GUID_0FE80B58_3E9E_4719_F47B_5DF4C24AC926'}
	(* Element-wise application of a bit-wise NOT operator to a container (integer only). *)
	FUNCTION F_VN_BitwiseNotContainer : HRESULT
	VAR_INPUT
		ipSrcContainer	:	ITcVnContainer;	(* Source container *)
		ipDestContainer	:	REFERENCE TO ITcVnContainer;	(* Returns the resulting container *)
		hrPrev	:	HRESULT;	(* HRESULT indicating the result of previous operations (If SUCCEEDED(hrPrev) equals false, no operation is executed.) *)
	END_VAR

END_FUNCTION

// Functions/Algebraic Container Operations/F_VN_BitwiseOrContainers

	{attribute 'TcIecLibraryType'}
	{attribute 'external_name' := 'F_VN_BitwiseOrContainers_GUID_088F9180_9532_479E_E411_693C42B6CCD5'}
	(* Element-wise application of a bit-wise OR operator to two containers (same length and type, integer only). *)
	FUNCTION F_VN_BitwiseOrContainers : HRESULT
	VAR_INPUT
		ipSrcContainer1	:	ITcVnContainer;	(* Source container 1 *)
		ipSrcContainer2	:	ITcVnContainer;	(* Source container 2 *)
		ipDestContainer	:	REFERENCE TO ITcVnContainer;	(* Returns the resulting container *)
		hrPrev	:	HRESULT;	(* HRESULT indicating the result of previous operations (If SUCCEEDED(hrPrev) equals false, no operation is executed.) *)
	END_VAR

END_FUNCTION

// Functions/Algebraic Container Operations/F_VN_BitwiseXorContainers

	{attribute 'TcIecLibraryType'}
	{attribute 'external_name' := 'F_VN_BitwiseXorContainers_GUID_48F66FE1_FBE7_4250_FEAC_4871DFC50E0D'}
	(* Element-wise application of a bit-wise XOR operator to two containers (same length and type, integer only). *)
	FUNCTION F_VN_BitwiseXorContainers : HRESULT
	VAR_INPUT
		ipSrcContainer1	:	ITcVnContainer;	(* Source container 1 *)
		ipSrcContainer2	:	ITcVnContainer;	(* Source container 2 *)
		ipDestContainer	:	REFERENCE TO ITcVnContainer;	(* Returns the resulting container *)
		hrPrev	:	HRESULT;	(* HRESULT indicating the result of previous operations (If SUCCEEDED(hrPrev) equals false, no operation is executed.) *)
	END_VAR

END_FUNCTION

// Functions/Algebraic Container Operations/F_VN_DivideContainers

	{attribute 'TcIecLibraryType'}
	{attribute 'external_name' := 'F_VN_DivideContainers_GUID_B7869534_57F7_4D38_E911_72B3E31E5756'}
	(* Element-wise division of two containers (same length and type). In case of integer division by zero, the resulting element is set to 0 and S_DIVISION_BY_ZERO is returned instead of S_OK (value can be changed in F_VN_DivideContainersExp). *)
	FUNCTION F_VN_DivideContainers : HRESULT
	VAR_INPUT
		ipSrcContainer1	:	ITcVnContainer;	(* Source container 1 *)
		ipSrcContainer2	:	ITcVnContainer;	(* Source container 2 *)
		ipDestContainer	:	REFERENCE TO ITcVnContainer;	(* Returns the resulting container *)
		hrPrev	:	HRESULT;	(* HRESULT indicating the result of previous operations (If SUCCEEDED(hrPrev) equals false, no operation is executed.) *)
	END_VAR

END_FUNCTION

// Functions/Algebraic Container Operations/F_VN_DivideContainersExp

	{attribute 'TcIecLibraryType'}
	{attribute 'external_name' := 'F_VN_DivideContainersExp_GUID_AF9B5326_9554_431A_D174_CE9CC4D0E21B'}
	(* Element-wise division of two containers (same length and type). In case of integer division by zero, the resulting element is set to nIntDivideByZeroResult and S_DIVISION_BY_ZERO is returned instead of S_OK. (expert function) *)
	FUNCTION F_VN_DivideContainersExp : HRESULT
	VAR_INPUT
		ipSrcContainer1	:	ITcVnContainer;	(* Source container 1 *)
		ipSrcContainer2	:	ITcVnContainer;	(* Source container 2 *)
		ipDestContainer	:	REFERENCE TO ITcVnContainer;	(* Returns the resulting container *)
		nIntDivideByZeroResult	:	LINT;	(* Value set as result in case of integer division by zero *)
		hrPrev	:	HRESULT;	(* HRESULT indicating the result of previous operations (If SUCCEEDED(hrPrev) equals false, no operation is executed.) *)
	END_VAR

END_FUNCTION

// Functions/Algebraic Container Operations/F_VN_MaxContainer

	{attribute 'TcIecLibraryType'}
	{attribute 'external_name' := 'F_VN_MaxContainer_GUID_7F1BFB8B_4BA4_4173_E808_A40C556A4EFC'}
	(* Element-wise maximum of two containers (same length and type). *)
	FUNCTION F_VN_MaxContainer : HRESULT
	VAR_INPUT
		ipSrcContainer1	:	ITcVnContainer;	(* Source container 1 *)
		ipSrcContainer2	:	ITcVnContainer;	(* Source container 2 *)
		ipDestContainer	:	REFERENCE TO ITcVnContainer;	(* Returns the resulting container *)
		hrPrev	:	HRESULT;	(* HRESULT indicating the result of previous operations (If SUCCEEDED(hrPrev) equals false, no operation is executed.) *)
	END_VAR

END_FUNCTION

// Functions/Algebraic Container Operations/F_VN_MinContainer

	{attribute 'TcIecLibraryType'}
	{attribute 'external_name' := 'F_VN_MinContainer_GUID_F57A6209_AE0C_4713_D3CA_8F1D8FFEC0C8'}
	(* Element-wise minimum of two containers (same length and type). *)
	FUNCTION F_VN_MinContainer : HRESULT
	VAR_INPUT
		ipSrcContainer1	:	ITcVnContainer;	(* Source container 1 *)
		ipSrcContainer2	:	ITcVnContainer;	(* Source container 2 *)
		ipDestContainer	:	REFERENCE TO ITcVnContainer;	(* Returns the resulting container *)
		hrPrev	:	HRESULT;	(* HRESULT indicating the result of previous operations (If SUCCEEDED(hrPrev) equals false, no operation is executed.) *)
	END_VAR

END_FUNCTION

// Functions/Algebraic Container Operations/F_VN_MultiplyContainers

	{attribute 'TcIecLibraryType'}
	{attribute 'external_name' := 'F_VN_MultiplyContainers_GUID_EDC07D82_2B29_43D7_E952_86C844E4756D'}
	(* Element-wise multiplication of two containers (same length and type). *)
	FUNCTION F_VN_MultiplyContainers : HRESULT
	VAR_INPUT
		ipSrcContainer1	:	ITcVnContainer;	(* Source container 1 *)
		ipSrcContainer2	:	ITcVnContainer;	(* Source container 2 *)
		ipDestContainer	:	REFERENCE TO ITcVnContainer;	(* Returns the resulting container *)
		hrPrev	:	HRESULT;	(* HRESULT indicating the result of previous operations (If SUCCEEDED(hrPrev) equals false, no operation is executed.) *)
	END_VAR

END_FUNCTION

// Functions/Algebraic Container Operations/F_VN_MultiplyWithContainerElements1

	{attribute 'TcIecLibraryType'}
	{attribute 'external_name' := 'F_VN_MultiplyWithContainerElements1_GUID_C2BF368D_3F5D_4387_FACE_116DE91F0C28'}
	(* Multiply each container element with a value. *)
	FUNCTION F_VN_MultiplyWithContainerElements1 : HRESULT
	VAR_INPUT
		fValue	:	LREAL;	(* Value *)
		ipContainer	:	ITcVnContainer;	(* Container with 1-dimensional elements *)
		hrPrev	:	HRESULT;	(* HRESULT indicating the result of previous operations (If SUCCEEDED(hrPrev) equals false, no operation is executed.) *)
	END_VAR

END_FUNCTION

// Functions/Algebraic Container Operations/F_VN_MultiplyWithContainerElements2

	{attribute 'TcIecLibraryType'}
	{attribute 'external_name' := 'F_VN_MultiplyWithContainerElements2_GUID_4FCDE80A_A060_4C3F_DA67_8A8C5682B9D5'}
	(* Multiply each container element with a value. *)
	FUNCTION F_VN_MultiplyWithContainerElements2 : HRESULT
	VAR_IN_OUT
		aValue	:	TcVnVector2_LREAL;	(* Value *)
	END_VAR
	VAR_INPUT
		ipContainer	:	ITcVnContainer;	(* Container with 2-dimensional elements *)
		hrPrev	:	HRESULT;	(* HRESULT indicating the result of previous operations (If SUCCEEDED(hrPrev) equals false, no operation is executed.) *)
	END_VAR

END_FUNCTION

// Functions/Algebraic Container Operations/F_VN_MultiplyWithContainerElements3

	{attribute 'TcIecLibraryType'}
	{attribute 'external_name' := 'F_VN_MultiplyWithContainerElements3_GUID_E4AA5061_0640_440C_D63F_C4AE31EC6028'}
	(* Multiply each container element with a value. *)
	FUNCTION F_VN_MultiplyWithContainerElements3 : HRESULT
	VAR_IN_OUT
		aValue	:	TcVnVector3_LREAL;	(* Value *)
	END_VAR
	VAR_INPUT
		ipContainer	:	ITcVnContainer;	(* Container with 3-dimensional elements *)
		hrPrev	:	HRESULT;	(* HRESULT indicating the result of previous operations (If SUCCEEDED(hrPrev) equals false, no operation is executed.) *)
	END_VAR

END_FUNCTION

// Functions/Algebraic Container Operations/F_VN_MultiplyWithContainerElements4

	{attribute 'TcIecLibraryType'}
	{attribute 'external_name' := 'F_VN_MultiplyWithContainerElements4_GUID_25796F55_FFA9_4C88_D1EE_4E25F01F1DC0'}
	(* Multiply each container element with a value. *)
	FUNCTION F_VN_MultiplyWithContainerElements4 : HRESULT
	VAR_IN_OUT
		aValue	:	TcVnVector4_LREAL;	(* Value *)
	END_VAR
	VAR_INPUT
		ipContainer	:	ITcVnContainer;	(* Container with 4-dimensional elements *)
		hrPrev	:	HRESULT;	(* HRESULT indicating the result of previous operations (If SUCCEEDED(hrPrev) equals false, no operation is executed.) *)
	END_VAR

END_FUNCTION

// Functions/Algebraic Container Operations/F_VN_NegateContainer

	{attribute 'TcIecLibraryType'}
	{attribute 'external_name' := 'F_VN_NegateContainer_GUID_FF195641_42B5_48AF_F8F8_0444DF37016B'}
	(* Element-wise negation of a container (two's complement). *)
	FUNCTION F_VN_NegateContainer : HRESULT
	VAR_INPUT
		ipSrcContainer	:	ITcVnContainer;	(* Source container *)
		ipDestContainer	:	REFERENCE TO ITcVnContainer;	(* Returns the resulting container (same type as ipSrcContainer) *)
		hrPrev	:	HRESULT;	(* HRESULT indicating the result of previous operations (If SUCCEEDED(hrPrev) equals false, no operation is executed.) *)
	END_VAR

END_FUNCTION

// Functions/Algebraic Container Operations/F_VN_SubtractContainers

	{attribute 'TcIecLibraryType'}
	{attribute 'external_name' := 'F_VN_SubtractContainers_GUID_D5559FDE_B583_41C0_E59D_45F7C831AD22'}
	(* Element-wise subtraction of two containers (same length and type). *)
	FUNCTION F_VN_SubtractContainers : HRESULT
	VAR_INPUT
		ipSrcContainer1	:	ITcVnContainer;	(* Source container 1 *)
		ipSrcContainer2	:	ITcVnContainer;	(* Source container 2 *)
		ipDestContainer	:	REFERENCE TO ITcVnContainer;	(* Returns the resulting container *)
		hrPrev	:	HRESULT;	(* HRESULT indicating the result of previous operations (If SUCCEEDED(hrPrev) equals false, no operation is executed.) *)
	END_VAR

END_FUNCTION

// Functions/Algebraic Image Operations/F_VN_AddImages

	{attribute 'TcIecLibraryType'}
	{attribute 'external_name' := 'F_VN_AddImages_GUID_9C3690A7_4C30_42AB_C7AC_F1A8E67F318F'}
	(* Element-wise addition of two images using saturation arithmetics. *)
	FUNCTION F_VN_AddImages : HRESULT
	VAR_INPUT
		ipSrcImage1	:	ITcVnImage;	(* First source image *)
		ipSrcImage2	:	ITcVnImage;	(* Second source image *)
		ipDestImage	:	REFERENCE TO ITcVnImage;	(* Destination image (An appropriate destination image will be created if required.) *)
		hrPrev	:	HRESULT;	(* HRESULT indicating the result of previous operations (If SUCCEEDED(hrPrev) equals false, no operation is executed.) *)
	END_VAR

END_FUNCTION

// Functions/Algebraic Image Operations/F_VN_AddImagesWeighted

	{attribute 'TcIecLibraryType'}
	{attribute 'external_name' := 'F_VN_AddImagesWeighted_GUID_90A66877_F045_48BF_CE26_998F4AE089DF'}
	(* Weighted, element-wise addition of two images using saturation arithmetics. *)
	FUNCTION F_VN_AddImagesWeighted : HRESULT
	VAR_INPUT
		ipSrcImage1	:	ITcVnImage;	(* First source image *)
		ipSrcImage2	:	ITcVnImage;	(* Second source image *)
		ipDestImage	:	REFERENCE TO ITcVnImage;	(* Destination image (An appropriate destination image will be created if required.) *)
		fWeight1	:	LREAL;	(* Weight factor applied to ipSrcImage1 *)
		fWeight2	:	LREAL;	(* Weight factor applied to ipSrcImage2 *)
		fDelta	:	LREAL;	(* Value added to the weighted sum of both images *)
		hrPrev	:	HRESULT;	(* HRESULT indicating the result of previous operations (If SUCCEEDED(hrPrev) equals false, no operation is executed.) *)
	END_VAR

END_FUNCTION

// Functions/Algebraic Image Operations/F_VN_AddImagesWeightedExp

	{attribute 'TcIecLibraryType'}
	{attribute 'external_name' := 'F_VN_AddImagesWeightedExp_GUID_4C622179_0696_4B9C_F08D_3B0F6FC7771C'}
	(* Weighted, element-wise addition of two images using saturation arithmetics. *)
	FUNCTION F_VN_AddImagesWeightedExp : HRESULT
	VAR_INPUT
		ipSrcImage1	:	ITcVnImage;	(* First source image *)
		ipSrcImage2	:	ITcVnImage;	(* Second source image *)
		ipDestImage	:	REFERENCE TO ITcVnImage;	(* Destination image (An appropriate destination image will be created if required.) *)
		fWeight1	:	LREAL;	(* Weight factor applied to ipSrcImage1 *)
		fWeight2	:	LREAL;	(* Weight factor applied to ipSrcImage2 *)
		fDelta	:	LREAL;	(* Value added to the weighted sum of both images *)
		eDestType	:	ETcVnElementType;	(* Destination image depth *)
		hrPrev	:	HRESULT;	(* HRESULT indicating the result of previous operations (If SUCCEEDED(hrPrev) equals false, no operation is executed.) *)
	END_VAR

END_FUNCTION

// Functions/Algebraic Image Operations/F_VN_AddScalarToImage

	{attribute 'TcIecLibraryType'}
	{attribute 'external_name' := 'F_VN_AddScalarToImage_GUID_B0F34FD6_06C2_426C_D311_E6F71C10C8A3'}
	(* Add a scalar value to each image pixel using saturation arithmetics. *)
	FUNCTION F_VN_AddScalarToImage : HRESULT
	VAR_INPUT
		fScalar	:	LREAL;	(* Scalar value *)
		ipSrcImage	:	ITcVnImage;	(* Source image *)
		ipDestImage	:	REFERENCE TO ITcVnImage;	(* Destination image (An appropriate destination image will be created if required.) *)
		hrPrev	:	HRESULT;	(* HRESULT indicating the result of previous operations (If SUCCEEDED(hrPrev) equals false, no operation is executed.) *)
	END_VAR

END_FUNCTION

// Functions/Algebraic Image Operations/F_VN_AddVectorToImage

	{attribute 'TcIecLibraryType'}
	{attribute 'external_name' := 'F_VN_AddVectorToImage_GUID_258467C2_CFCB_47AE_D0D0_1B5809CC6321'}
	(* Add a vector (1 element for each image channel) to each image pixel using saturation arithmetics. *)
	FUNCTION F_VN_AddVectorToImage : HRESULT
	VAR_IN_OUT
		aVector	:	TcVnVector4_LREAL;	(* 4-element vector (1 element for each image channel. If the image has less channels, the further vector elements are ignored.) *)
	END_VAR
	VAR_INPUT
		ipSrcImage	:	ITcVnImage;	(* Source image *)
		ipDestImage	:	REFERENCE TO ITcVnImage;	(* Destination image (An appropriate destination image will be created if required.) *)
		hrPrev	:	HRESULT;	(* HRESULT indicating the result of previous operations (If SUCCEEDED(hrPrev) equals false, no operation is executed.) *)
	END_VAR

END_FUNCTION

// Functions/Algebraic Image Operations/F_VN_BitwiseAndImages

	{attribute 'TcIecLibraryType'}
	{attribute 'external_name' := 'F_VN_BitwiseAndImages_GUID_462FD49F_1A04_491C_CC36_BE1D063F9860'}
	(* Element-wise application of a bit-wise AND operator to two images. *)
	FUNCTION F_VN_BitwiseAndImages : HRESULT
	VAR_INPUT
		ipSrcImage1	:	ITcVnImage;	(* First source image *)
		ipSrcImage2	:	ITcVnImage;	(* Second source image *)
		ipDestImage	:	REFERENCE TO ITcVnImage;	(* Destination image (An appropriate destination image will be created if required.) *)
		hrPrev	:	HRESULT;	(* HRESULT indicating the result of previous operations (If SUCCEEDED(hrPrev) equals false, no operation is executed.) *)
	END_VAR

END_FUNCTION

// Functions/Algebraic Image Operations/F_VN_BitwiseAndImagesExp

	{attribute 'TcIecLibraryType'}
	{attribute 'external_name' := 'F_VN_BitwiseAndImagesExp_GUID_D0D56EAF_2010_4A14_F9FA_BBC8768F6F87'}
	(* Element-wise application of a bit-wise AND operator to two images. (expert function) *)
	FUNCTION F_VN_BitwiseAndImagesExp : HRESULT
	VAR_INPUT
		ipSrcImage1	:	ITcVnImage;	(* First source image *)
		ipSrcImage2	:	ITcVnImage;	(* Second source image *)
		ipDestImage	:	REFERENCE TO ITcVnImage;	(* Destination image (An appropriate destination image will be created if required.) *)
		ipMask	:	ITcVnImage;	(* Mask to limit the operation to specific pixel positions (mask value 0: skip pixel, mask value > 0: apply operation to pixel) *)
		hrPrev	:	HRESULT;	(* HRESULT indicating the result of previous operations (If SUCCEEDED(hrPrev) equals false, no operation is executed.) *)
	END_VAR

END_FUNCTION

// Functions/Algebraic Image Operations/F_VN_BitwiseAndScalarWithImage

	{attribute 'TcIecLibraryType'}
	{attribute 'external_name' := 'F_VN_BitwiseAndScalarWithImage_GUID_C0A3C3C3_3169_4652_DF99_BB129581A1C8'}
	(* Bitwise and a scalar value with each image pixel. *)
	FUNCTION F_VN_BitwiseAndScalarWithImage : HRESULT
	VAR_INPUT
		fScalar	:	LREAL;	(* Scalar value *)
		ipSrcImage	:	ITcVnImage;	(* Source image *)
		ipDestImage	:	REFERENCE TO ITcVnImage;	(* Destination image (An appropriate destination image will be created if required.) *)
		hrPrev	:	HRESULT;	(* HRESULT indicating the result of previous operations (If SUCCEEDED(hrPrev) equals false, no operation is executed.) *)
	END_VAR

END_FUNCTION

// Functions/Algebraic Image Operations/F_VN_BitwiseAndVectorWithImage

	{attribute 'TcIecLibraryType'}
	{attribute 'external_name' := 'F_VN_BitwiseAndVectorWithImage_GUID_C46F8886_8C53_4F79_E07D_F90B3BD58931'}
	(* Bitwise and a vector (1 element for each image channel) with each image pixel. *)
	FUNCTION F_VN_BitwiseAndVectorWithImage : HRESULT
	VAR_IN_OUT
		aVector	:	TcVnVector4_LREAL;	(* 4-element vector (1 element for each image channel. If the image has less channels, the further vector elements are ignored.) *)
	END_VAR
	VAR_INPUT
		ipSrcImage	:	ITcVnImage;	(* Source image *)
		ipDestImage	:	REFERENCE TO ITcVnImage;	(* Destination image (An appropriate destination image will be created if required.) *)
		hrPrev	:	HRESULT;	(* HRESULT indicating the result of previous operations (If SUCCEEDED(hrPrev) equals false, no operation is executed.) *)
	END_VAR

END_FUNCTION

// Functions/Algebraic Image Operations/F_VN_BitwiseNotImage

	{attribute 'TcIecLibraryType'}
	{attribute 'external_name' := 'F_VN_BitwiseNotImage_GUID_FC99E208_B709_446C_C9B3_7FF4420977D5'}
	(* Element-wise application of a bit-wise NOT operator to an image. *)
	FUNCTION F_VN_BitwiseNotImage : HRESULT
	VAR_INPUT
		ipSrcImage	:	ITcVnImage;	(* Source image *)
		ipDestImage	:	REFERENCE TO ITcVnImage;	(* Destination image (An appropriate destination image will be created if required.) *)
		hrPrev	:	HRESULT;	(* HRESULT indicating the result of previous operations (If SUCCEEDED(hrPrev) equals false, no operation is executed.) *)
	END_VAR

END_FUNCTION

// Functions/Algebraic Image Operations/F_VN_BitwiseNotImageExp

	{attribute 'TcIecLibraryType'}
	{attribute 'external_name' := 'F_VN_BitwiseNotImageExp_GUID_C2E609D0_C935_4BFE_FC3C_E4D71DC4DE46'}
	(* Element-wise application of a bit-wise NOT operator to an image. (expert function) *)
	FUNCTION F_VN_BitwiseNotImageExp : HRESULT
	VAR_INPUT
		ipSrcImage	:	ITcVnImage;	(* Source image *)
		ipDestImage	:	REFERENCE TO ITcVnImage;	(* Destination image (An appropriate destination image will be created if required.) *)
		ipMask	:	ITcVnImage;	(* Mask to limit the operation to specific pixel positions (mask value 0: skip pixel, mask value > 0: apply operation to pixel) *)
		hrPrev	:	HRESULT;	(* HRESULT indicating the result of previous operations (If SUCCEEDED(hrPrev) equals false, no operation is executed.) *)
	END_VAR

END_FUNCTION

// Functions/Algebraic Image Operations/F_VN_BitwiseOrImages

	{attribute 'TcIecLibraryType'}
	{attribute 'external_name' := 'F_VN_BitwiseOrImages_GUID_3134DBBB_571C_4608_ED08_011D919A7B11'}
	(* Element-wise application of a bit-wise OR operator to two images. *)
	FUNCTION F_VN_BitwiseOrImages : HRESULT
	VAR_INPUT
		ipSrcImage1	:	ITcVnImage;	(* First source image *)
		ipSrcImage2	:	ITcVnImage;	(* Second source image *)
		ipDestImage	:	REFERENCE TO ITcVnImage;	(* Destination image (An appropriate destination image will be created if required.) *)
		hrPrev	:	HRESULT;	(* HRESULT indicating the result of previous operations (If SUCCEEDED(hrPrev) equals false, no operation is executed.) *)
	END_VAR

END_FUNCTION

// Functions/Algebraic Image Operations/F_VN_BitwiseOrImagesExp

	{attribute 'TcIecLibraryType'}
	{attribute 'external_name' := 'F_VN_BitwiseOrImagesExp_GUID_9D7A3554_D1EF_4AB1_E62E_F6B2AC222B1C'}
	(* Element-wise application of a bit-wise OR operator to two images. (expert function) *)
	FUNCTION F_VN_BitwiseOrImagesExp : HRESULT
	VAR_INPUT
		ipSrcImage1	:	ITcVnImage;	(* First source image *)
		ipSrcImage2	:	ITcVnImage;	(* Second source image *)
		ipDestImage	:	REFERENCE TO ITcVnImage;	(* Destination image (An appropriate destination image will be created if required.) *)
		ipMask	:	ITcVnImage;	(* Mask to limit the operation to specific pixel positions (mask value 0: skip pixel, mask value > 0: apply operation to pixel) *)
		hrPrev	:	HRESULT;	(* HRESULT indicating the result of previous operations (If SUCCEEDED(hrPrev) equals false, no operation is executed.) *)
	END_VAR

END_FUNCTION

// Functions/Algebraic Image Operations/F_VN_BitwiseOrScalarWithImage

	{attribute 'TcIecLibraryType'}
	{attribute 'external_name' := 'F_VN_BitwiseOrScalarWithImage_GUID_F7B1578C_D8F8_451F_FA12_B51CB639AC9B'}
	(* Bitwise or a scalar value with each image pixel. *)
	FUNCTION F_VN_BitwiseOrScalarWithImage : HRESULT
	VAR_INPUT
		fScalar	:	LREAL;	(* Scalar value *)
		ipSrcImage	:	ITcVnImage;	(* Source image *)
		ipDestImage	:	REFERENCE TO ITcVnImage;	(* Destination image (An appropriate destination image will be created if required.) *)
		hrPrev	:	HRESULT;	(* HRESULT indicating the result of previous operations (If SUCCEEDED(hrPrev) equals false, no operation is executed.) *)
	END_VAR

END_FUNCTION

// Functions/Algebraic Image Operations/F_VN_BitwiseOrVectorWithImage

	{attribute 'TcIecLibraryType'}
	{attribute 'external_name' := 'F_VN_BitwiseOrVectorWithImage_GUID_B069D285_0262_4843_D8EC_29854617293E'}
	(* Bitwise or a vector (1 element for each image channel) with each image pixel. *)
	FUNCTION F_VN_BitwiseOrVectorWithImage : HRESULT
	VAR_IN_OUT
		aVector	:	TcVnVector4_LREAL;	(* 4-element vector (1 element for each image channel. If the image has less channels, the further vector elements are ignored.) *)
	END_VAR
	VAR_INPUT
		ipSrcImage	:	ITcVnImage;	(* Source image *)
		ipDestImage	:	REFERENCE TO ITcVnImage;	(* Destination image (An appropriate destination image will be created if required.) *)
		hrPrev	:	HRESULT;	(* HRESULT indicating the result of previous operations (If SUCCEEDED(hrPrev) equals false, no operation is executed.) *)
	END_VAR

END_FUNCTION

// Functions/Algebraic Image Operations/F_VN_BitwiseXorImages

	{attribute 'TcIecLibraryType'}
	{attribute 'external_name' := 'F_VN_BitwiseXorImages_GUID_F08CDDF1_A51E_467C_E70B_25674FC950C4'}
	(* Element-wise application of a bit-wise XOR operator to two images. *)
	FUNCTION F_VN_BitwiseXorImages : HRESULT
	VAR_INPUT
		ipSrcImage1	:	ITcVnImage;	(* First source image *)
		ipSrcImage2	:	ITcVnImage;	(* Second source image *)
		ipDestImage	:	REFERENCE TO ITcVnImage;	(* Destination image (An appropriate destination image will be created if required.) *)
		hrPrev	:	HRESULT;	(* HRESULT indicating the result of previous operations (If SUCCEEDED(hrPrev) equals false, no operation is executed.) *)
	END_VAR

END_FUNCTION

// Functions/Algebraic Image Operations/F_VN_BitwiseXorImagesExp

	{attribute 'TcIecLibraryType'}
	{attribute 'external_name' := 'F_VN_BitwiseXorImagesExp_GUID_A3CD730B_E417_4068_D2E8_4F522103EE15'}
	(* Element-wise application of a bit-wise XOR operator to two images. (expert function) *)
	FUNCTION F_VN_BitwiseXorImagesExp : HRESULT
	VAR_INPUT
		ipSrcImage1	:	ITcVnImage;	(* First source image *)
		ipSrcImage2	:	ITcVnImage;	(* Second source image *)
		ipDestImage	:	REFERENCE TO ITcVnImage;	(* Destination image (An appropriate destination image will be created if required.) *)
		ipMask	:	ITcVnImage;	(* Mask to limit the operation to specific pixel positions (mask value 0: skip pixel, mask value > 0: apply operation to pixel) *)
		hrPrev	:	HRESULT;	(* HRESULT indicating the result of previous operations (If SUCCEEDED(hrPrev) equals false, no operation is executed.) *)
	END_VAR

END_FUNCTION

// Functions/Algebraic Image Operations/F_VN_BitwiseXorScalarWithImage

	{attribute 'TcIecLibraryType'}
	{attribute 'external_name' := 'F_VN_BitwiseXorScalarWithImage_GUID_C9489A65_3E8A_410F_C0E2_8420600EB87A'}
	(* Bitwise xor a scalar value with each image pixel. *)
	FUNCTION F_VN_BitwiseXorScalarWithImage : HRESULT
	VAR_INPUT
		fScalar	:	LREAL;	(* Scalar value *)
		ipSrcImage	:	ITcVnImage;	(* Source image *)
		ipDestImage	:	REFERENCE TO ITcVnImage;	(* Destination image (An appropriate destination image will be created if required.) *)
		hrPrev	:	HRESULT;	(* HRESULT indicating the result of previous operations (If SUCCEEDED(hrPrev) equals false, no operation is executed.) *)
	END_VAR

END_FUNCTION

// Functions/Algebraic Image Operations/F_VN_BitwiseXorVectorWithImage

	{attribute 'TcIecLibraryType'}
	{attribute 'external_name' := 'F_VN_BitwiseXorVectorWithImage_GUID_4F3E278F_B38D_4193_C4A8_82EFD40C045D'}
	(* Bitwise xor a vector (1 element for each image channel) with each image pixel. *)
	FUNCTION F_VN_BitwiseXorVectorWithImage : HRESULT
	VAR_IN_OUT
		aVector	:	TcVnVector4_LREAL;	(* 4-element vector (1 element for each image channel. If the image has less channels, the further vector elements are ignored.) *)
	END_VAR
	VAR_INPUT
		ipSrcImage	:	ITcVnImage;	(* Source image *)
		ipDestImage	:	REFERENCE TO ITcVnImage;	(* Destination image (An appropriate destination image will be created if required.) *)
		hrPrev	:	HRESULT;	(* HRESULT indicating the result of previous operations (If SUCCEEDED(hrPrev) equals false, no operation is executed.) *)
	END_VAR

END_FUNCTION

// Functions/Algebraic Image Operations/F_VN_BlendImages

	{attribute 'TcIecLibraryType'}
	{attribute 'external_name' := 'F_VN_BlendImages_GUID_21C63199_32BD_4107_F987_066B2811244D'}
	(* Blends two images, i.e. dest = (src1 * weight1 + src2 * weight2) / (weight1 + weight2). *)
	FUNCTION F_VN_BlendImages : HRESULT
	VAR_INPUT
		ipSrcImage1	:	ITcVnImage;	(* First source image (ET_USINT or ET_REAL) *)
		ipSrcImage2	:	ITcVnImage;	(* Second source image (same type and size as ipSrcImage1) *)
		ipWeights1	:	ITcVnImage;	(* Weights for ipSrcImage1 (1 channel, ET_REAL) *)
		ipWeights2	:	ITcVnImage;	(* Weights for ipSrcImage2 (1 channel, ET_REAL) *)
		ipDestImage	:	REFERENCE TO ITcVnImage;	(* Destination image (An appropriate destination image will be created if required.) *)
		hrPrev	:	HRESULT;	(* HRESULT indicating the result of previous operations (If SUCCEEDED(hrPrev) equals false, no operation is executed.) *)
	END_VAR

END_FUNCTION

// Functions/Algebraic Image Operations/F_VN_DivideImageByScalar

	{attribute 'TcIecLibraryType'}
	{attribute 'external_name' := 'F_VN_DivideImageByScalar_GUID_E0840C81_C1F8_4EE9_F3EB_BB42E4839093'}
	(* Divide each image pixel by a scalar value using saturation arithmetics. *)
	FUNCTION F_VN_DivideImageByScalar : HRESULT
	VAR_INPUT
		ipSrcImage	:	ITcVnImage;	(* Source image *)
		fScalar	:	LREAL;	(* Scalar value *)
		ipDestImage	:	REFERENCE TO ITcVnImage;	(* Destination image (An appropriate destination image will be created if required.) *)
		hrPrev	:	HRESULT;	(* HRESULT indicating the result of previous operations (If SUCCEEDED(hrPrev) equals false, no operation is executed.) *)
	END_VAR

END_FUNCTION

// Functions/Algebraic Image Operations/F_VN_DivideImageByVector

	{attribute 'TcIecLibraryType'}
	{attribute 'external_name' := 'F_VN_DivideImageByVector_GUID_107BF212_B17E_435F_F136_78890960AFDB'}
	(* Divides each image pixel by a vector (1 element for each image channel) using saturation arithmetics. *)
	FUNCTION F_VN_DivideImageByVector : HRESULT
	VAR_INPUT
		ipSrcImage	:	ITcVnImage;	(* Source image *)
	END_VAR
	VAR_IN_OUT
		aVector	:	TcVnVector4_LREAL;	(* 4-element vector (1 element for each image channel. If the image has less channels, the further vector elements are ignored.) *)
	END_VAR
	VAR_INPUT
		ipDestImage	:	REFERENCE TO ITcVnImage;	(* Destination image (An appropriate destination image will be created if required.) *)
		hrPrev	:	HRESULT;	(* HRESULT indicating the result of previous operations (If SUCCEEDED(hrPrev) equals false, no operation is executed.) *)
	END_VAR

END_FUNCTION

// Functions/Algebraic Image Operations/F_VN_DivideImages

	{attribute 'TcIecLibraryType'}
	{attribute 'external_name' := 'F_VN_DivideImages_GUID_F08F50B9_3B3D_47DC_FCE9_0221DB136AE5'}
	(* Element-wise division of two images using saturation arithmetics. (A division by zero equals zero.) *)
	FUNCTION F_VN_DivideImages : HRESULT
	VAR_INPUT
		ipSrcImage1	:	ITcVnImage;	(* First source image (dividend) *)
		ipSrcImage2	:	ITcVnImage;	(* Second source image (divisor) *)
		ipDestImage	:	REFERENCE TO ITcVnImage;	(* Destination image (An appropriate destination image will be created if required.) *)
		hrPrev	:	HRESULT;	(* HRESULT indicating the result of previous operations (If SUCCEEDED(hrPrev) equals false, no operation is executed.) *)
	END_VAR

END_FUNCTION

// Functions/Algebraic Image Operations/F_VN_DivideScalarByImage

	{attribute 'TcIecLibraryType'}
	{attribute 'external_name' := 'F_VN_DivideScalarByImage_GUID_A3FA6C84_F52E_4B0C_C141_7106EFC170B2'}
	(* Divides a scalar value by each image pixel using saturation arithmetics. *)
	FUNCTION F_VN_DivideScalarByImage : HRESULT
	VAR_INPUT
		fScalar	:	LREAL;	(* Scalar value *)
		ipSrcImage	:	ITcVnImage;	(* Source image *)
		ipDestImage	:	REFERENCE TO ITcVnImage;	(* Destination image (An appropriate destination image will be created if required.) *)
		hrPrev	:	HRESULT;	(* HRESULT indicating the result of previous operations (If SUCCEEDED(hrPrev) equals false, no operation is executed.) *)
	END_VAR

END_FUNCTION

// Functions/Algebraic Image Operations/F_VN_DivideVectorByImage

	{attribute 'TcIecLibraryType'}
	{attribute 'external_name' := 'F_VN_DivideVectorByImage_GUID_A8DF0FE9_C3E0_4F0A_F10C_371750F1AD2A'}
	(* Divides a vector (1 element for each image channel) by each image pixel using saturation arithmetics. *)
	FUNCTION F_VN_DivideVectorByImage : HRESULT
	VAR_IN_OUT
		aVector	:	TcVnVector4_LREAL;	(* 4-element vector (1 element for each image channel. If the image has less channels, the further vector elements are ignored.) *)
	END_VAR
	VAR_INPUT
		ipSrcImage	:	ITcVnImage;	(* Source image *)
		ipDestImage	:	REFERENCE TO ITcVnImage;	(* Destination image (An appropriate destination image will be created if required.) *)
		hrPrev	:	HRESULT;	(* HRESULT indicating the result of previous operations (If SUCCEEDED(hrPrev) equals false, no operation is executed.) *)
	END_VAR

END_FUNCTION

// Functions/Algebraic Image Operations/F_VN_ElementwiseExp

	{attribute 'TcIecLibraryType'}
	{attribute 'external_name' := 'F_VN_ElementwiseExp_GUID_8A34D5F3_DD4F_4FD9_F7CD_DCC1EB94D033'}
	(* Computes the natural exponent of each pixel value. *)
	FUNCTION F_VN_ElementwiseExp : HRESULT
	VAR_INPUT
		ipSrcImage	:	ITcVnImage;	(* Source image (REAL or LREAL) *)
		ipDestImage	:	REFERENCE TO ITcVnImage;	(* Destination image (Same type and size as ipSrcImage, an appropriate image will be created if required.) *)
		hrPrev	:	HRESULT;	(* HRESULT indicating the result of previous operations (If SUCCEEDED(hrPrev) equals false, no operation is executed.) *)
	END_VAR

END_FUNCTION

// Functions/Algebraic Image Operations/F_VN_ElementwiseLog

	{attribute 'TcIecLibraryType'}
	{attribute 'external_name' := 'F_VN_ElementwiseLog_GUID_92E3CFCA_7FE0_49C7_CE79_11AB977F927A'}
	(* Computes the natural logarithm of each pixel value. *)
	FUNCTION F_VN_ElementwiseLog : HRESULT
	VAR_INPUT
		ipSrcImage	:	ITcVnImage;	(* Source image (REAL or LREAL) *)
		ipDestImage	:	REFERENCE TO ITcVnImage;	(* Destination image (Same type and size as ipSrcImage, an appropriate image will be created if required.) *)
		hrPrev	:	HRESULT;	(* HRESULT indicating the result of previous operations (If SUCCEEDED(hrPrev) equals false, no operation is executed.) *)
	END_VAR

END_FUNCTION

// Functions/Algebraic Image Operations/F_VN_MaxImage

	{attribute 'TcIecLibraryType'}
	{attribute 'external_name' := 'F_VN_MaxImage_GUID_F2AA4AAA_21FB_4D33_CDD0_138266A8FC1F'}
	(* Element-wise maximum of two images. *)
	FUNCTION F_VN_MaxImage : HRESULT
	VAR_INPUT
		ipSrcImage1	:	ITcVnImage;	(* First source image *)
		ipSrcImage2	:	ITcVnImage;	(* Second source image *)
		ipDestImage	:	REFERENCE TO ITcVnImage;	(* Destination image (An appropriate destination image will be created if required.) *)
		hrPrev	:	HRESULT;	(* HRESULT indicating the result of previous operations (If SUCCEEDED(hrPrev) equals false, no operation is executed.) *)
	END_VAR

END_FUNCTION

// Functions/Algebraic Image Operations/F_VN_MaxImageExp

	{attribute 'TcIecLibraryType'}
	{attribute 'external_name' := 'F_VN_MaxImageExp_GUID_FCE7DFB7_EBCA_46F1_EA15_BDD38EFCCCC7'}
	(* Element-wise maximum of two images. (expert function) *)
	FUNCTION F_VN_MaxImageExp : HRESULT
	VAR_INPUT
		ipSrcImage1	:	ITcVnImage;	(* First source image *)
		ipSrcImage2	:	ITcVnImage;	(* Second source image *)
		ipDestImage	:	REFERENCE TO ITcVnImage;	(* Destination image (An appropriate destination image will be created if required.) *)
		ipMask	:	ITcVnImage;	(* Mask of type USINT *)
		hrPrev	:	HRESULT;	(* HRESULT indicating the result of previous operations (If SUCCEEDED(hrPrev) equals false, no operation is executed.) *)
	END_VAR

END_FUNCTION

// Functions/Algebraic Image Operations/F_VN_MaxImageWithScalar

	{attribute 'TcIecLibraryType'}
	{attribute 'external_name' := 'F_VN_MaxImageWithScalar_GUID_A76A3E5D_83D1_4146_FB57_692C87DC60CB'}
	(* Element-wise maximum of image and scalar value. *)
	FUNCTION F_VN_MaxImageWithScalar : HRESULT
	VAR_INPUT
		fScalar	:	LREAL;	(* Scalar value *)
		ipSrcImage	:	ITcVnImage;	(* Source image *)
		ipDestImage	:	REFERENCE TO ITcVnImage;	(* Destination image (An appropriate destination image will be created if required.) *)
		hrPrev	:	HRESULT;	(* HRESULT indicating the result of previous operations (If SUCCEEDED(hrPrev) equals false, no operation is executed.) *)
	END_VAR

END_FUNCTION

// Functions/Algebraic Image Operations/F_VN_MaxImageWithScalarExp

	{attribute 'TcIecLibraryType'}
	{attribute 'external_name' := 'F_VN_MaxImageWithScalarExp_GUID_D7599590_6C53_4F86_FD3F_E0393A5B8959'}
	(* Element-wise maximum of image and scalar value. (expert function) *)
	FUNCTION F_VN_MaxImageWithScalarExp : HRESULT
	VAR_INPUT
		fScalar	:	LREAL;	(* Scalar value *)
		ipSrcImage	:	ITcVnImage;	(* Source image *)
		ipDestImage	:	REFERENCE TO ITcVnImage;	(* Destination image (An appropriate destination image will be created if required.) *)
		ipMask	:	ITcVnImage;	(* Mask of type USINT *)
		hrPrev	:	HRESULT;	(* HRESULT indicating the result of previous operations (If SUCCEEDED(hrPrev) equals false, no operation is executed.) *)
	END_VAR

END_FUNCTION

// Functions/Algebraic Image Operations/F_VN_MaxImageWithVector

	{attribute 'TcIecLibraryType'}
	{attribute 'external_name' := 'F_VN_MaxImageWithVector_GUID_451BB152_500D_4604_E3F5_DEFC3C132AA8'}
	(* Element-wise maximum of image and vector (1 element for each image channel). *)
	FUNCTION F_VN_MaxImageWithVector : HRESULT
	VAR_IN_OUT
		aVector	:	TcVnVector4_LREAL;	(* 4-element vector (1 element for each image channel. If the image has less channels, the further vector elements are ignored.) *)
	END_VAR
	VAR_INPUT
		ipSrcImage	:	ITcVnImage;	(* Source image *)
		ipDestImage	:	REFERENCE TO ITcVnImage;	(* Destination image (An appropriate destination image will be created if required.) *)
		hrPrev	:	HRESULT;	(* HRESULT indicating the result of previous operations (If SUCCEEDED(hrPrev) equals false, no operation is executed.) *)
	END_VAR

END_FUNCTION

// Functions/Algebraic Image Operations/F_VN_MaxImageWithVectorExp

	{attribute 'TcIecLibraryType'}
	{attribute 'external_name' := 'F_VN_MaxImageWithVectorExp_GUID_55F6D290_CF4D_4C6E_E281_120207851D67'}
	(* Element-wise maximum of image and vector (1 element for each image channel). (expert function) *)
	FUNCTION F_VN_MaxImageWithVectorExp : HRESULT
	VAR_IN_OUT
		aVector	:	TcVnVector4_LREAL;	(* 4-element vector (1 element for each image channel. If the image has less channels, the further vector elements are ignored.) *)
	END_VAR
	VAR_INPUT
		ipSrcImage	:	ITcVnImage;	(* Source image *)
		ipDestImage	:	REFERENCE TO ITcVnImage;	(* Destination image (An appropriate destination image will be created if required.) *)
		ipMask	:	ITcVnImage;	(* Mask of type USINT *)
		hrPrev	:	HRESULT;	(* HRESULT indicating the result of previous operations (If SUCCEEDED(hrPrev) equals false, no operation is executed.) *)
	END_VAR

END_FUNCTION

// Functions/Algebraic Image Operations/F_VN_MinImage

	{attribute 'TcIecLibraryType'}
	{attribute 'external_name' := 'F_VN_MinImage_GUID_923261CE_7C20_4377_E691_323AC849D3F8'}
	(* Element-wise minimum of two images. *)
	FUNCTION F_VN_MinImage : HRESULT
	VAR_INPUT
		ipSrcImage1	:	ITcVnImage;	(* First source image *)
		ipSrcImage2	:	ITcVnImage;	(* Second source image *)
		ipDestImage	:	REFERENCE TO ITcVnImage;	(* Destination image (An appropriate destination image will be created if required.) *)
		hrPrev	:	HRESULT;	(* HRESULT indicating the result of previous operations (If SUCCEEDED(hrPrev) equals false, no operation is executed.) *)
	END_VAR

END_FUNCTION

// Functions/Algebraic Image Operations/F_VN_MinImageExp

	{attribute 'TcIecLibraryType'}
	{attribute 'external_name' := 'F_VN_MinImageExp_GUID_76F3BAE0_02F0_462B_D3D8_4C5E0FF60550'}
	(* Element-wise minimum of two images. (expert function) *)
	FUNCTION F_VN_MinImageExp : HRESULT
	VAR_INPUT
		ipSrcImage1	:	ITcVnImage;	(* First source image *)
		ipSrcImage2	:	ITcVnImage;	(* Second source image *)
		ipDestImage	:	REFERENCE TO ITcVnImage;	(* Destination image (An appropriate destination image will be created if required.) *)
		ipMask	:	ITcVnImage;	(* Mask of type USINT *)
		hrPrev	:	HRESULT;	(* HRESULT indicating the result of previous operations (If SUCCEEDED(hrPrev) equals false, no operation is executed.) *)
	END_VAR

END_FUNCTION

// Functions/Algebraic Image Operations/F_VN_MinImageWithScalar

	{attribute 'TcIecLibraryType'}
	{attribute 'external_name' := 'F_VN_MinImageWithScalar_GUID_7FEB738E_CE2F_456A_CE7A_2983AD11DCED'}
	(* Element-wise minimum of image and scalar value. *)
	FUNCTION F_VN_MinImageWithScalar : HRESULT
	VAR_INPUT
		fScalar	:	LREAL;	(* Scalar value *)
		ipSrcImage	:	ITcVnImage;	(* Source image *)
		ipDestImage	:	REFERENCE TO ITcVnImage;	(* Destination image (An appropriate destination image will be created if required.) *)
		hrPrev	:	HRESULT;	(* HRESULT indicating the result of previous operations (If SUCCEEDED(hrPrev) equals false, no operation is executed.) *)
	END_VAR

END_FUNCTION

// Functions/Algebraic Image Operations/F_VN_MinImageWithScalarExp

	{attribute 'TcIecLibraryType'}
	{attribute 'external_name' := 'F_VN_MinImageWithScalarExp_GUID_BAFC74CD_46B2_4946_CFD0_AEA7CC35B7A8'}
	(* Element-wise minimum of image and scalar value. (expert function) *)
	FUNCTION F_VN_MinImageWithScalarExp : HRESULT
	VAR_INPUT
		fScalar	:	LREAL;	(* Scalar value *)
		ipSrcImage	:	ITcVnImage;	(* Source image *)
		ipDestImage	:	REFERENCE TO ITcVnImage;	(* Destination image (An appropriate destination image will be created if required.) *)
		ipMask	:	ITcVnImage;	(* Mask of type USINT *)
		hrPrev	:	HRESULT;	(* HRESULT indicating the result of previous operations (If SUCCEEDED(hrPrev) equals false, no operation is executed.) *)
	END_VAR

END_FUNCTION

// Functions/Algebraic Image Operations/F_VN_MinImageWithVector

	{attribute 'TcIecLibraryType'}
	{attribute 'external_name' := 'F_VN_MinImageWithVector_GUID_5E26309F_DD89_40DF_D825_D27522210737'}
	(* Element-wise minimum of image and vector (1 element for each image channel). *)
	FUNCTION F_VN_MinImageWithVector : HRESULT
	VAR_IN_OUT
		aVector	:	TcVnVector4_LREAL;	(* 4-element vector (1 element for each image channel. If the image has less channels, the further vector elements are ignored.) *)
	END_VAR
	VAR_INPUT
		ipSrcImage	:	ITcVnImage;	(* Source image *)
		ipDestImage	:	REFERENCE TO ITcVnImage;	(* Destination image (An appropriate destination image will be created if required.) *)
		hrPrev	:	HRESULT;	(* HRESULT indicating the result of previous operations (If SUCCEEDED(hrPrev) equals false, no operation is executed.) *)
	END_VAR

END_FUNCTION

// Functions/Algebraic Image Operations/F_VN_MinImageWithVectorExp

	{attribute 'TcIecLibraryType'}
	{attribute 'external_name' := 'F_VN_MinImageWithVectorExp_GUID_F149B716_5A59_4CA5_EC7E_5572681B0822'}
	(* Element-wise minimum of image and vector (1 element for each image channel). (expert function) *)
	FUNCTION F_VN_MinImageWithVectorExp : HRESULT
	VAR_IN_OUT
		aVector	:	TcVnVector4_LREAL;	(* 4-element vector (1 element for each image channel. If the image has less channels, the further vector elements are ignored.) *)
	END_VAR
	VAR_INPUT
		ipSrcImage	:	ITcVnImage;	(* Source image *)
		ipDestImage	:	REFERENCE TO ITcVnImage;	(* Destination image (An appropriate destination image will be created if required.) *)
		ipMask	:	ITcVnImage;	(* Mask of type USINT *)
		hrPrev	:	HRESULT;	(* HRESULT indicating the result of previous operations (If SUCCEEDED(hrPrev) equals false, no operation is executed.) *)
	END_VAR

END_FUNCTION

// Functions/Algebraic Image Operations/F_VN_MultiplyImages

	{attribute 'TcIecLibraryType'}
	{attribute 'external_name' := 'F_VN_MultiplyImages_GUID_018144D7_9EF9_4D08_E1AC_2F66435404D7'}
	(* Element-wise multiplication of two images using saturation arithmetics. *)
	FUNCTION F_VN_MultiplyImages : HRESULT
	VAR_INPUT
		ipSrcImage1	:	ITcVnImage;	(* First source image *)
		ipSrcImage2	:	ITcVnImage;	(* Second source image *)
		ipDestImage	:	REFERENCE TO ITcVnImage;	(* Destination image (An appropriate destination image will be created if required.) *)
		hrPrev	:	HRESULT;	(* HRESULT indicating the result of previous operations (If SUCCEEDED(hrPrev) equals false, no operation is executed.) *)
	END_VAR

END_FUNCTION

// Functions/Algebraic Image Operations/F_VN_MultiplyImageWithScalar

	{attribute 'TcIecLibraryType'}
	{attribute 'external_name' := 'F_VN_MultiplyImageWithScalar_GUID_32003E64_4658_416E_FD2A_08BF723BCDD6'}
	(* Multiply each image pixel by a scalar value using saturation arithmetics. *)
	FUNCTION F_VN_MultiplyImageWithScalar : HRESULT
	VAR_INPUT
		fScalar	:	LREAL;	(* Scalar value *)
		ipSrcImage	:	ITcVnImage;	(* Source image *)
		ipDestImage	:	REFERENCE TO ITcVnImage;	(* Destination image (An appropriate destination image will be created if required.) *)
		hrPrev	:	HRESULT;	(* HRESULT indicating the result of previous operations (If SUCCEEDED(hrPrev) equals false, no operation is executed.) *)
	END_VAR

END_FUNCTION

// Functions/Algebraic Image Operations/F_VN_MultiplyImageWithVector

	{attribute 'TcIecLibraryType'}
	{attribute 'external_name' := 'F_VN_MultiplyImageWithVector_GUID_D97DB062_280E_463C_CA5F_8961AD43078E'}
	(* Multiply each image pixel by a vector (1 element for each image channel) using saturation arithmetics. *)
	FUNCTION F_VN_MultiplyImageWithVector : HRESULT
	VAR_IN_OUT
		aVector	:	TcVnVector4_LREAL;	(* 4-element vector (1 element for each image channel. If the image has less channels, the further vector elements are ignored.) *)
	END_VAR
	VAR_INPUT
		ipSrcImage	:	ITcVnImage;	(* Source image *)
		ipDestImage	:	REFERENCE TO ITcVnImage;	(* Destination image (An appropriate destination image will be created if required.) *)
		hrPrev	:	HRESULT;	(* HRESULT indicating the result of previous operations (If SUCCEEDED(hrPrev) equals false, no operation is executed.) *)
	END_VAR

END_FUNCTION

// Functions/Algebraic Image Operations/F_VN_SubtractImageFromScalar

	{attribute 'TcIecLibraryType'}
	{attribute 'external_name' := 'F_VN_SubtractImageFromScalar_GUID_3B813E9C_3037_43D6_CE6C_28B258C921AD'}
	(* Subtract each image pixel from a scalar value using saturation arithmetics. *)
	FUNCTION F_VN_SubtractImageFromScalar : HRESULT
	VAR_INPUT
		fScalar	:	LREAL;	(* Scalar value *)
		ipSrcImage	:	ITcVnImage;	(* Source image *)
		ipDestImage	:	REFERENCE TO ITcVnImage;	(* Destination image (An appropriate destination image will be created if required.) *)
		hrPrev	:	HRESULT;	(* HRESULT indicating the result of previous operations (If SUCCEEDED(hrPrev) equals false, no operation is executed.) *)
	END_VAR

END_FUNCTION

// Functions/Algebraic Image Operations/F_VN_SubtractImageFromVector

	{attribute 'TcIecLibraryType'}
	{attribute 'external_name' := 'F_VN_SubtractImageFromVector_GUID_947A63A3_D271_4F29_DF18_FF9EA9DC7468'}
	(* Subtract each image pixel from a vector (1 element for each image channel) using saturation arithmetics. *)
	FUNCTION F_VN_SubtractImageFromVector : HRESULT
	VAR_IN_OUT
		aVector	:	TcVnVector4_LREAL;	(* 4-element vector (1 element for each image channel. If the image has less channels, the further vector elements are ignored.) *)
	END_VAR
	VAR_INPUT
		ipSrcImage	:	ITcVnImage;	(* Source image *)
		ipDestImage	:	REFERENCE TO ITcVnImage;	(* Destination image (An appropriate destination image will be created if required.) *)
		hrPrev	:	HRESULT;	(* HRESULT indicating the result of previous operations (If SUCCEEDED(hrPrev) equals false, no operation is executed.) *)
	END_VAR

END_FUNCTION

// Functions/Algebraic Image Operations/F_VN_SubtractImages

	{attribute 'TcIecLibraryType'}
	{attribute 'external_name' := 'F_VN_SubtractImages_GUID_1080354C_2BCC_4BB4_CDC2_6FAB0E80307B'}
	(* Element-wise subtraction of two images using saturation arithmetics. *)
	FUNCTION F_VN_SubtractImages : HRESULT
	VAR_INPUT
		ipSrcImage1	:	ITcVnImage;	(* First source image (minuend) *)
		ipSrcImage2	:	ITcVnImage;	(* Second source image (subtrahend) *)
		ipDestImage	:	REFERENCE TO ITcVnImage;	(* Destination image (An appropriate destination image will be created if required.) *)
		hrPrev	:	HRESULT;	(* HRESULT indicating the result of previous operations (If SUCCEEDED(hrPrev) equals false, no operation is executed.) *)
	END_VAR

END_FUNCTION

// Functions/Algebraic Image Operations/F_VN_SubtractScalarFromImage

	{attribute 'TcIecLibraryType'}
	{attribute 'external_name' := 'F_VN_SubtractScalarFromImage_GUID_C95ED9CB_1D4B_42F8_D283_FBB42A767E8F'}
	(* Subtract a scalar value from each image pixel using saturation arithmetics. *)
	FUNCTION F_VN_SubtractScalarFromImage : HRESULT
	VAR_INPUT
		ipSrcImage	:	ITcVnImage;	(* Source image *)
		fScalar	:	LREAL;	(* Scalar value *)
		ipDestImage	:	REFERENCE TO ITcVnImage;	(* Destination image (An appropriate destination image will be created if required.) *)
		hrPrev	:	HRESULT;	(* HRESULT indicating the result of previous operations (If SUCCEEDED(hrPrev) equals false, no operation is executed.) *)
	END_VAR

END_FUNCTION

// Functions/Algebraic Image Operations/F_VN_SubtractVectorFromImage

	{attribute 'TcIecLibraryType'}
	{attribute 'external_name' := 'F_VN_SubtractVectorFromImage_GUID_B96E11E7_A362_417F_D4C1_B898BCA14AF4'}
	(* Subtract a vector (1 element for each image channel) from each image pixel using saturation arithmetics. *)
	FUNCTION F_VN_SubtractVectorFromImage : HRESULT
	VAR_INPUT
		ipSrcImage	:	ITcVnImage;	(* Source image *)
	END_VAR
	VAR_IN_OUT
		aVector	:	TcVnVector4_LREAL;	(* 4-element vector (1 element for each image channel. If the image has less channels, the further vector elements are ignored.) *)
	END_VAR
	VAR_INPUT
		ipDestImage	:	REFERENCE TO ITcVnImage;	(* Destination image (An appropriate destination image will be created if required.) *)
		hrPrev	:	HRESULT;	(* HRESULT indicating the result of previous operations (If SUCCEEDED(hrPrev) equals false, no operation is executed.) *)
	END_VAR

END_FUNCTION

// Functions/Image Analysis/F_VN_CannyEdgeDetection

	{attribute 'TcIecLibraryType'}
	{attribute 'external_name' := 'F_VN_CannyEdgeDetection_GUID_2E7A680F_A16F_445C_D68E_80E989C197BA'}
	(* Find edges using the Canny edge detection algorithm. *)
	FUNCTION F_VN_CannyEdgeDetection : HRESULT
	VAR_INPUT
		ipSrcImage	:	ITcVnImage;	(* Source image (elements of type USINT) *)
		ipDestImage	:	REFERENCE TO ITcVnImage;	(* Destination image (elements of type USINT. An appropriate destination image will be created if required.) *)
		fThresholdLow	:	LREAL;	(* Low threshold *)
		fThresholdHigh	:	LREAL;	(* High threshold *)
		hrPrev	:	HRESULT;	(* HRESULT indicating the result of previous operations (If SUCCEEDED(hrPrev) equals false, no operation is executed.) *)
	END_VAR

END_FUNCTION

// Functions/Image Analysis/F_VN_CannyEdgeDetectionExp

	{attribute 'TcIecLibraryType'}
	{attribute 'external_name' := 'F_VN_CannyEdgeDetectionExp_GUID_EE23BD2D_50C1_413A_E097_5B0937F81AD4'}
	(* Find edges using the Canny edge detection algorithm. (expert function) *)
	FUNCTION F_VN_CannyEdgeDetectionExp : HRESULT
	VAR_INPUT
		ipSrcImage	:	ITcVnImage;	(* Source image (elements of type USINT) *)
		ipDestImage	:	REFERENCE TO ITcVnImage;	(* Destination image (elements of type USINT. An appropriate destination image will be created if required.) *)
		fThresholdLow	:	LREAL;	(* Low threshold *)
		fThresholdHigh	:	LREAL;	(* High threshold *)
		nApertureSize	:	UDINT;	(* Aperture size for the Sobel operator (3, 5, 7) *)
		bL2Gradient	:	BOOL;	(* If true, the more accurate (and slower) L2 norm is used instead of the L1 norm *)
		hrPrev	:	HRESULT;	(* HRESULT indicating the result of previous operations (If SUCCEEDED(hrPrev) equals false, no operation is executed.) *)
	END_VAR

END_FUNCTION

// Functions/Image Analysis/F_VN_ConnectedComponents

	{attribute 'TcIecLibraryType'}
	{attribute 'external_name' := 'F_VN_ConnectedComponents_GUID_E0B0C8B9_C8D4_4A4A_CB1C_413A9FA46C8B'}
	(* Computes the connected components of an image. *)
	FUNCTION F_VN_ConnectedComponents : HRESULT
	VAR_INPUT
		ipSrcImage	:	ITcVnImage;	(* Source image (USINT, 1 channel, binary) *)
		ipLabelImage	:	REFERENCE TO ITcVnImage;	(* Returns the labels for each source image pixel (1 channel, DINT. An appropriate destination image will be created if required.) *)
	END_VAR
	VAR_IN_OUT
		nLabels	:	DINT;	(* Returns the number of labels *)
	END_VAR
	VAR_INPUT
		hrPrev	:	HRESULT;	(* HRESULT indicating the result of previous operations (If SUCCEEDED(hrPrev) equals false, no operation is executed.) *)
	END_VAR

END_FUNCTION

// Functions/Image Analysis/F_VN_ConnectedComponentsExp

	{attribute 'TcIecLibraryType'}
	{attribute 'external_name' := 'F_VN_ConnectedComponentsExp_GUID_382D6AE8_26CB_48FA_C95A_16017B284AF7'}
	(* Computes the connected components of an image. (expert function) *)
	FUNCTION F_VN_ConnectedComponentsExp : HRESULT
	VAR_INPUT
		ipSrcImage	:	ITcVnImage;	(* Source image (USINT, 1 channel, binary) *)
		ipLabelImage	:	REFERENCE TO ITcVnImage;	(* Returns the labels for each source image pixel (1 channel, type depends on eLabelType. An appropriate destination image will be created if required.) *)
	END_VAR
	VAR_IN_OUT
		nLabels	:	DINT;	(* Returns the number of labels *)
	END_VAR
	VAR_INPUT
		eConnectivity	:	ETcVnPixelConnectivity;	(* Selects if 4- or 8-way pixel connectivity should be used *)
		eLabelType	:	ETcVnElementType;	(* Selects the type of ipLabelImage (only UINT or DINT supported) *)
		eAlgorithm	:	ETcVnConnectedComponentsAlgorithm;	(* Selects the applied algorithm *)
		hrPrev	:	HRESULT;	(* HRESULT indicating the result of previous operations (If SUCCEEDED(hrPrev) equals false, no operation is executed.) *)
	END_VAR

END_FUNCTION

// Functions/Image Analysis/F_VN_ConnectedComponentsWithStats

	{attribute 'TcIecLibraryType'}
	{attribute 'external_name' := 'F_VN_ConnectedComponentsWithStats_GUID_8EF45095_6CC6_42A9_C9EC_792C56477083'}
	(* Computes the connected components and corresponding statistics of an image. *)
	FUNCTION F_VN_ConnectedComponentsWithStats : HRESULT
	VAR_INPUT
		ipSrcImage	:	ITcVnImage;	(* Source image (USINT, 1 channel, binary) *)
		ipLabelImage	:	REFERENCE TO ITcVnImage;	(* Returns the labels for each source image pixel (1 channel, DINT. An appropriate destination image will be created if required.) *)
		ipBoundingBoxes	:	REFERENCE TO ITcVnContainer;	(* Returns the bounding boxes for each labeled region. (ContainerType_Vector_TcVnRectangle_DINT; Non-zero interface pointers are reused.) *)
		ipNumPixels	:	REFERENCE TO ITcVnContainer;	(* Returns the number of pixels for each labeled region. (ContainerType_Vector_DINT; Non-zero interface pointers are reused.) *)
		ipCentroids	:	REFERENCE TO ITcVnContainer;	(* Returns the centroids for each labeled region. (ContainerType_Vector_TcVnPoint2_LREAL; Non-zero interface pointers are reused.) *)
	END_VAR
	VAR_IN_OUT
		nLabels	:	DINT;	(* Returns the number of labels *)
	END_VAR
	VAR_INPUT
		hrPrev	:	HRESULT;	(* HRESULT indicating the result of previous operations (If SUCCEEDED(hrPrev) equals false, no operation is executed.) *)
	END_VAR

END_FUNCTION

// Functions/Image Analysis/F_VN_ConnectedComponentsWithStatsExp

	{attribute 'TcIecLibraryType'}
	{attribute 'external_name' := 'F_VN_ConnectedComponentsWithStatsExp_GUID_46E2F003_6D91_4C47_EA72_776E6555D3FB'}
	(* Computes the connected components and corresponding statistics of an image. (expert function) *)
	FUNCTION F_VN_ConnectedComponentsWithStatsExp : HRESULT
	VAR_INPUT
		ipSrcImage	:	ITcVnImage;	(* Source image (USINT, 1 channel, binary) *)
		ipLabelImage	:	REFERENCE TO ITcVnImage;	(* Returns the labels for each source image pixel (1 channel, DINT. An appropriate destination image will be created if required.) *)
		ipBoundingBoxes	:	REFERENCE TO ITcVnContainer;	(* Returns the bounding boxes for each labeled region. (ContainerType_Vector_TcVnRectangle_DINT; Non-zero interface pointers are reused.) *)
		ipNumPixels	:	REFERENCE TO ITcVnContainer;	(* Returns the number of pixels for each labeled region. (ContainerType_Vector_DINT; Non-zero interface pointers are reused.) *)
		ipCentroids	:	REFERENCE TO ITcVnContainer;	(* Returns the centroids for each labeled region. (ContainerType_Vector_TcVnPoint2_LREAL; Non-zero interface pointers are reused.) *)
	END_VAR
	VAR_IN_OUT
		nLabels	:	DINT;	(* Returns the number of labels *)
	END_VAR
	VAR_INPUT
		eConnectivity	:	ETcVnPixelConnectivity;	(* Selects if 4- or 8-way pixel connectivity should be used *)
		eLabelType	:	ETcVnElementType;	(* Selects the type of ipLabelImage (only UINT or DINT supported) *)
		eAlgorithm	:	ETcVnConnectedComponentsAlgorithm;	(* Selects the applied algorithm *)
		hrPrev	:	HRESULT;	(* HRESULT indicating the result of previous operations (If SUCCEEDED(hrPrev) equals false, no operation is executed.) *)
	END_VAR

END_FUNCTION

// Functions/Image Analysis/F_VN_CountNonZeroPixels

	{attribute 'TcIecLibraryType'}
	{attribute 'external_name' := 'F_VN_CountNonZeroPixels_GUID_1E0CCDA6_F7C3_40BD_DA4A_181037AC1F45'}
	(* Counts the non-zero pixels in a single-channel image (e.g. useful to analyze threshold results). *)
	FUNCTION F_VN_CountNonZeroPixels : HRESULT
	VAR_INPUT
		ipSrcImage	:	ITcVnImage;	(* Source image (1 channel) *)
	END_VAR
	VAR_IN_OUT
		nNonZero	:	ULINT;	(* Returns the number of non-zero pixels in ipSrcImage *)
	END_VAR
	VAR_INPUT
		hrPrev	:	HRESULT;	(* HRESULT indicating the result of previous operations (If SUCCEEDED(hrPrev) equals false, no operation is executed.) *)
	END_VAR

END_FUNCTION

// Functions/Image Analysis/F_VN_DistanceTransformation

	{attribute 'TcIecLibraryType'}
	{attribute 'external_name' := 'F_VN_DistanceTransformation_GUID_CDB18E62_66B1_4107_E135_A12986D9C9DE'}
	(* Calculates the distance transformation, which is the distance to the closest zero pixel in a binary image. *)
	FUNCTION F_VN_DistanceTransformation : HRESULT
	VAR_INPUT
		ipSrcImage	:	ITcVnImage;	(* Source image (USINT, 1 channel) *)
		ipDestImage	:	REFERENCE TO ITcVnImage;	(* Destination image (REAL, 1 channel. An appropriate destination image will be created if required.) *)
		eDistanceType	:	ETcVnDistanceType;	(* Distance computation method (supported: L1, L2, C) *)
		eMaskSize	:	ETcVnDistanceTransformationMask;	(* Size of the distance transformation mask *)
		hrPrev	:	HRESULT;	(* HRESULT indicating the result of previous operations (If SUCCEEDED(hrPrev) equals false, no operation is executed.) *)
	END_VAR

END_FUNCTION

// Functions/Image Analysis/F_VN_DistanceTransformationExp

	{attribute 'TcIecLibraryType'}
	{attribute 'external_name' := 'F_VN_DistanceTransformationExp_GUID_CFD62F8F_5AD5_4028_D0B8_60D21D9E0BCC'}
	(* Calculates the distance transformation, which is the distance to the closest zero pixel in a binary image. Additionally, an image with component labels is created (discrete Voronoi diagram). (expert function) *)
	FUNCTION F_VN_DistanceTransformationExp : HRESULT
	VAR_INPUT
		ipSrcImage	:	ITcVnImage;	(* Source image (USINT, 1 channel) *)
		ipDestImage	:	REFERENCE TO ITcVnImage;	(* Destination image (REAL, 1 channel. An appropriate destination image will be created if required.) *)
		eDistanceType	:	ETcVnDistanceType;	(* Distance computation method (supported: L1, L2, C) *)
		eMaskSize	:	ETcVnDistanceTransformationMask;	(* Size of the distance transformation mask (PRECISE not supported for label computation) *)
		ipDestLabels	:	REFERENCE TO ITcVnImage;	(* Returns the component labels (Discrete Voronoi diagram; DINT, 1 channel. An appropriate image will be created if required.) *)
		eLabelType	:	ETcVnDistanceTransformationLabel;	(* Type of the labels *)
		hrPrev	:	HRESULT;	(* HRESULT indicating the result of previous operations (If SUCCEEDED(hrPrev) equals false, no operation is executed.) *)
	END_VAR

END_FUNCTION

// Functions/Image Analysis/F_VN_GetConnectedComponent

	{attribute 'TcIecLibraryType'}
	{attribute 'external_name' := 'F_VN_GetConnectedComponent_GUID_A1A9BF7E_233D_406B_F8AB_27E356FE4E44'}
	(* Get the mask image of a connected component from a label image based on the label ID. *)
	FUNCTION F_VN_GetConnectedComponent : HRESULT
	VAR_INPUT
		ipLabelImage	:	ITcVnImage;	(* Image containing labels for each pixel (1 channel DINT or UINT). *)
		nLabelID	:	DINT;	(* Value of the requested label *)
		ipMaskImage	:	REFERENCE TO ITcVnImage;	(* Returns a mask image marking the pixels that belong to the component (1 channel USINT.) *)
		hrPrev	:	HRESULT;	(* HRESULT indicating the result of previous operations (If SUCCEEDED(hrPrev) equals false, no operation is executed.) *)
	END_VAR

END_FUNCTION

// Functions/Image Analysis/F_VN_GetConnectedComponentExp

	{attribute 'TcIecLibraryType'}
	{attribute 'external_name' := 'F_VN_GetConnectedComponentExp_GUID_18409C68_BA0F_4DEB_D486_971CD7B84334'}
	(* Get the mask image (and optionally the outer contour) of a connected component from a label image based on the label ID. (expert function) *)
	FUNCTION F_VN_GetConnectedComponentExp : HRESULT
	VAR_INPUT
		ipLabelImage	:	ITcVnImage;	(* Image containing labels for each pixel (1 channel DINT or UINT). *)
		nLabelID	:	DINT;	(* Value of the requested label *)
		ipMaskImage	:	REFERENCE TO ITcVnImage;	(* Returns a mask image marking the pixels that belong to the component (1 channel USINT. Mask is optional, set to 0 if not required.) *)
		ipContourPoints	:	REFERENCE TO ITcVnContainer;	(* Returns the outer contour of the component(ContainerType_Vector_TcVnPoint2_DINT. Contour is optional, set to 0 if not required.) *)
		hrPrev	:	HRESULT;	(* HRESULT indicating the result of previous operations (If SUCCEEDED(hrPrev) equals false, no operation is executed.) *)
	END_VAR

END_FUNCTION

// Functions/Image Analysis/F_VN_ImageAbsoluteAverage

	{attribute 'TcIecLibraryType'}
	{attribute 'external_name' := 'F_VN_ImageAbsoluteAverage_GUID_5AB63B48_311C_407E_FD1D_1FB980C384BA'}
	(* Computes the average absolute pixel value of an image. *)
	FUNCTION F_VN_ImageAbsoluteAverage : HRESULT
	VAR_INPUT
		ipSrcImage	:	ITcVnImage;	(* Source image *)
	END_VAR
	VAR_IN_OUT
		fAverage	:	LREAL;	(* Returns the average absolute pixel value *)
	END_VAR
	VAR_INPUT
		hrPrev	:	HRESULT;	(* HRESULT indicating the result of previous operations (If SUCCEEDED(hrPrev) equals false, no operation is executed.) *)
	END_VAR

END_FUNCTION

// Functions/Image Analysis/F_VN_ImageAverage

	{attribute 'TcIecLibraryType'}
	{attribute 'external_name' := 'F_VN_ImageAverage_GUID_8EE9A1FA_8FFD_42B5_E175_F3A205B9F7DB'}
	(* Computes the (channel-wise) average pixel value of an image. *)
	FUNCTION F_VN_ImageAverage : HRESULT
	VAR_INPUT
		ipSrcImage	:	ITcVnImage;	(* Source image (1 - 4 channels) *)
	END_VAR
	VAR_IN_OUT
		aAverage	:	TcVnVector4_LREAL;	(* Returns the (channel-wise) average pixel value of ipSrcImage *)
	END_VAR
	VAR_INPUT
		hrPrev	:	HRESULT;	(* HRESULT indicating the result of previous operations (If SUCCEEDED(hrPrev) equals false, no operation is executed.) *)
	END_VAR

END_FUNCTION

// Functions/Image Analysis/F_VN_ImageAverageExp

	{attribute 'TcIecLibraryType'}
	{attribute 'external_name' := 'F_VN_ImageAverageExp_GUID_4EBF4B4E_76AA_4A10_C0FA_EE1CC39B6EA0'}
	(* Computes the (channel-wise) average pixel value of an image. (expert function) *)
	FUNCTION F_VN_ImageAverageExp : HRESULT
	VAR_INPUT
		ipSrcImage	:	ITcVnImage;	(* Source image (1 - 4 channels) *)
	END_VAR
	VAR_IN_OUT
		aAverage	:	TcVnVector4_LREAL;	(* Returns the (channel-wise) average pixel value of ipSrcImage *)
	END_VAR
	VAR_INPUT
		ipMask	:	ITcVnImage;	(* Mask of type USINT (1 channel) *)
		hrPrev	:	HRESULT;	(* HRESULT indicating the result of previous operations (If SUCCEEDED(hrPrev) equals false, no operation is executed.) *)
	END_VAR

END_FUNCTION

// Functions/Image Analysis/F_VN_ImageAverageStdDev

	{attribute 'TcIecLibraryType'}
	{attribute 'external_name' := 'F_VN_ImageAverageStdDev_GUID_B92DA123_C708_4459_E4AB_8724C8CF9EEF'}
	(* Computes the (channel-wise) average pixel value and the corresponding standard deviation of an image. *)
	FUNCTION F_VN_ImageAverageStdDev : HRESULT
	VAR_INPUT
		ipSrcImage	:	ITcVnImage;	(* Source image (1 - 4 channels) *)
	END_VAR
	VAR_IN_OUT
		aAverage	:	TcVnVector4_LREAL;	(* Returns the (channel-wise) average pixel value of ipSrcImage *)
		aStdDev	:	TcVnVector4_LREAL;	(* Returns the (channel-wise) pixel value standard deviation of ipSrcImage *)
	END_VAR
	VAR_INPUT
		hrPrev	:	HRESULT;	(* HRESULT indicating the result of previous operations (If SUCCEEDED(hrPrev) equals false, no operation is executed.) *)
	END_VAR

END_FUNCTION

// Functions/Image Analysis/F_VN_ImageAverageStdDevExp

